// TwinCAT 3 PLC project PLC1
// Title: Sample Demo-Rack
// Company: Beckhoff Automation GmbH & Co. KG
// Author: Michael Golz
// ProjectVersion: 1.0.0
// ProgramVersion: 3.1.4026.14
// libraries:
//   Standard, * (System)
//   Tc2_Drive, * (Beckhoff Automation GmbH)
//   Tc2_EtherCAT, * (Beckhoff Automation GmbH)
//   Tc2_IoFunctions, * (Beckhoff Automation GmbH)
//   Tc2_Math, * (Beckhoff Automation GmbH)
//   Tc2_MC2, * (Beckhoff Automation GmbH)
//   Tc2_MC2_Camming, * (Beckhoff Automation GmbH)
//   Tc2_MC2_Drive, * (Beckhoff Automation GmbH)
//   Tc2_MC2_XFC, * (Beckhoff Automation GmbH)
//   Tc2_NCI, * (Beckhoff Automation GmbH)
//   Tc2_NcKinematicTransformation, * (Beckhoff Automation GmbH)
//   Tc2_PlcInterpolation, * (Beckhoff Automation GmbH)
//   Tc2_Standard, * (Beckhoff Automation GmbH)
//   Tc2_SUPS, * (Beckhoff Automation GmbH)
//   Tc2_System, * (Beckhoff Automation GmbH)
//   Tc2_Utilities, * (Beckhoff Automation GmbH)
//   Tc3_Database, * (Beckhoff Automation GmbH)
//   Tc3_EventLogger, * (Beckhoff Automation GmbH)
//   Tc3_Interfaces, * (Beckhoff Automation GmbH)
//   Tc3_IotBase, * (Beckhoff Automation GmbH)
//   Tc3_JsonXml, * (Beckhoff Automation GmbH)
//   Tc3_Module, * (Beckhoff Automation GmbH)
//   Tc3_RealtimeMonitoring, * (Beckhoff Automation GmbH)
//   TwinSafe3Diagnostics_v0.2.3, * (Beckhoff Automation LLC - Sample Code)
//   VisuDialogs, * (System)
// project tree:
//   DUTs/00_MainBlocks/ E_SystemStartupSequence.TcDUT
//   DUTs/20_Axis/ E_AxisReversingSequence.TcDUT, E_McResetStatus.TcDUT
//   DUTs/30_EtherCatDiagnostic/ E_EcDiacStatus.TcDUT, E_EcGetSlaveName.TcDUT, E_EcSystemStatus.TcDUT, ST_EcTerminalDiagInfo.TcDUT
//   DUTs/40_TwinSAFE/ ST_AdsAddr.TcDUT
//   DUTs/40_TwinSAFE/TwinSAFE_Connection/AX5805/ E_TsDiagnosisObjektsFA10AX5805.TcDUT, E_TsErrIndicesFA82AX5805.TcDUT, ST_TsControlWordAX5805.TcDUT, ST_TsDiagObjectsFA10AX5805.TcDUT, ST_TsErrIndicesFA82AX5805.TcDUT, ST_TsStatusWordAX5805.TcDUT
//   DUTs/40_TwinSAFE/TwinSAFE_Connection/EK1914/ ST_TsDiagObjectsBitsEK1914.TcDUT, ST_TsDiagObjectsEK1914.TcDUT
//   DUTs/40_TwinSAFE/TwinSAFE_Connection/EL1904/ ST_TsDiagObjectsBitsEL1904.TcDUT, ST_TsDiagObjectsEL1904.TcDUT
//   DUTs/40_TwinSAFE/TwinSAFE_Connection/EL2904/ ST_TsDiagObjectsBitsEL2904.TcDUT, ST_TsDiagObjectsEL2904.TcDUT
//   DUTs/40_TwinSAFE/TwinSAFE_Connection/ E_TsCycleDiagObj.TcDUT, ST_TsConnectionInfo1Byte.TcDUT, ST_TsConnectionInfo2Byte.TcDUT, ST_TsConnectionInfo8Byte.TcDUT, ST_TsConnectionInfoEL3214.TcDUT, ST_TsConnectionInfoEL5021.TcDUT, ST_TsSlave2Temp.TcDUT, ST_TsSlave3Temp.TcDUT
//   DUTs/40_TwinSAFE/TwinSAFE_Functionblocks/ E_TsFbType.TcDUT, ST_TsFbInfo.TcDUT
//   DUTs/40_TwinSAFE/TwinSAFE_Group/ ST_TsGroupInfo.TcDUT
//   DUTs/ E_SampleMode.TcDUT
//   / extMarkTask.TcTTO, GlobalTextList.TcGTLO, PlcTask.TcTTO, PlcTaskFast.TcTTO, Visualization Manager.TcVMO (not stored)
//   GVLs/ GVL.TcGVL, GVL00_IO_CX.TcGVL, GVL01_IO_EK1100.TcGVL, GVL02_IO_EK1101.TcGVL, GVL10_VAR_PRG.TcGVL, GVL20_Axis.TcGVL, GVL30_DiagnosticEtherCAT.TcGVL
//   POUs/Motion/ CamTable.TcPOU, Ext_SP_Gen.TcPOU, Axis1.TcPOU, AxisGeneral.TcPOU, Axis2.TcPOU, Axis3.TcPOU, Axis4.TcPOU, NCI.TcPOU
//   POUs/Database Server/ CSVSample.TcPOU, E_WriteMode.TcDUT, FB_CSV_Access.TcPOU, ST_CSVDataStruct.TcDUT
//   POUs/GeneralPlcBlocks/ FB_GenerateData.TcPOU, Blinker.TcPOU, ClockGenerator.TcPOU, GeneralPlc.TcPOU
//   POUs/IoT and JsonXml/FBs/ FB_JSONEncoding.TcPOU, FB_MqttCom_String.TcPOU, prgPopulateStructure.TcPOU
//   POUs/IoT and JsonXml/ IoTDataStruct.TcDUT, IoT_JSON_XML.TcPOU
//   POUs/MainPOUs/ MAIN.TcPOU, MAINFast.TcPOU, V_MAIN.TcVIS
//   POUs/GeneralPlcBlocks/Components/ FB_Blinker.TcPOU, F_Scaling.TcPOU
//   POUs/Motion/Components/ FB_Axis.TcPOU, FB_AxisAX5xxx.TcPOU, FB_ReversingSequence.TcPOU, MC_Reset_Ax5xxx.TcPOU
//   POUs/EtherCatDiagnostic/Components/ FB_DiagnosticEtherCAT.TcPOU
//   POUs/EtherCatDiagnostic/ DiagnosticEtherCAT.TcPOU
//   POUs/RT Monitor/ extMarksPrg.TcPOU, simpleMarksPrg.TcPOU
//   POUs/RT Monitor/logging/ ConsumeTime.TcPOU
//   POUs/Sample OOP/Cylinder/ FB_Cylinder.TcPOU, FB_CylinderDiag.TcPOU, ICylinder.TcIO
//   POUs/Sample OOP/ FB_OOPAxisTable.TcPOU, FB_OOPCylinderRegulator.TcPOU
//   POUs/Sample OOP/Regulator/ FB_BasicP.TcPOU, FB_BasicPID.TcPOU, IRegulator.TcIO, ST_RegParams.TcDUT
//   POUs/Sample OOP/Table/Axis/ FB_AX5000Axis.TcPOU, FB_NcAxis.TcPOU, IAxis.TcIO
//   POUs/Sample OOP/Table/ E_AxisState.TcDUT, E_MoveCmd.TcDUT, FB_Table.TcPOU
//   POUs/TwinSAFE/Components/ FB_EcGetSlaveName.TcPOU, FB_TwinSafeConnectionAX5805.TcPOU, FB_TwinSafeConnectionEK1914.TcPOU, FB_TwinSafeConnectionEL1904.TcPOU, FB_TwinSafeConnectionEL2904.TcPOU, FB_TwinSafeConnectionEL3214.TcPOU, FB_TwinSafeConnectionEL5021.TcPOU, FB_TwinSafeFB.TcPOU, FB_TwinSafeGroup.TcPOU, FB_TwinSafeGroupExt.TcPOU
//   POUs/TwinSAFE/ TwinSAFE.TcPOU
//   POUs/XFC/ AverageOut.TcPOU, DcTimes.TcPOU, AnalogOutputOversampling.TcPOU, PositionCamTimeStampAxis2.TcPOU, SignalLengthMeasurementCamAxis2.TcPOU, TouchProbeTimeStampCamAxis2.TcPOU
//   POUs/Sample OOP Conveyor/Axis Blocks/ FB_AX5000.TcPOU, FB_AxisNc.TcPOU, FB_Stepper.TcPOU, FB_VeryBasicMotor.TcPOU, I_Axis.TcIO
//   POUs/Sample OOP Conveyor/Device And Station Blocks/ FB_Conveyor.TcPOU, FB_Device.TcPOU, FB_Station.TcPOU, FB_TransferStation.TcPOU, GVL_Products.TcGVL, I_Mode.TcIO
//   POUs/Sample OOP Conveyor/Device And Station Blocks/Internal/ E_Modes.TcDUT, E_PartQuality.TcDUT, ST_PartData.TcDUT
//   POUs/Sample OOP Conveyor/ FB_OOPConveyor.TcPOU, V_OOP_Conveyor.TcVIS
//   POUs/Sample OOP Conveyor/Internal Visus/ Conveyor.TcVIS, ConveyorAuto.TcVIS, ConveyorData.TcVIS
//   POUs/Sample UML SC/ FB_UML_SC_Composite.TcPOU, FB_UML_SC_Lamp.TcPOU, GVL_UML.TcGVL, Visu_Composite.TcVIS, Visu_Lamp.TcVIS
//   POUs/SampleIEC Languages/Datatypes/ E_Commands.TcDUT, E_Operation.TcDUT
//   POUs/SampleIEC Languages/FunctionBlocks/ FB_CFC_SamplePOU.TcPOU, FB_CFC_SamplePouPageOriented.TcPOU, FB_FBD_IL_LD_SamplePOU.TcPOU, FB_SFC_SamplePou.TcPOU, FB_ST_SamplePOU.TcPOU
//   POUs/SampleIEC Languages/ MAIN_CFC.TcPOU, MAIN_CFC_PageOriented.TcPOU, MAIN_FBD_IL_LD.TcPOU, MAIN_SFC.TcPOU, MAIN_ST.TcPOU
//   VISUs/ MotionProfiles.TcVIS, HmiEtherCatDiagnostic.TcVIS, HmiAxisReversingSequence.TcVIS, HmiStartPage.TcVIS, HmiTwinSAFEDiagnostic.TcVIS
//   VISUs/HmiTemplatesAxis/ TplAxisControl.TcVIS, TplAxisReversingSequence.TcVIS
//   VISUs/HmiTemplatesTwinSAFE/ TplTsConnectionAX5805.TcVIS, TplTsConnectionEK1914.TcVIS, TplTsConnectionEL1904.TcVIS, TplTsConnectionEL2904.TcVIS, TplTsConnectionEL3214.TcVIS, TplTsConnectionEL5021.TcVIS, TplTsFb.TcVIS, TplTsGroup.TcVIS, TplTsGroupExt.TcVIS
// real-time tasks:
//   TASK PlcTask: cycle T#1ms, priority 8, ADS port 350
//   TASK PlcTaskFast: cycle T#100us, priority 4, ADS port 351
//   TASK VISU_TASK: cycle T#200000us, priority 30, ADS port 352
//   TASK extMarkTask: cycle T#1ms, priority 20, ADS port 353
// motion (NC):
//   TASK NC-Task 1 SAF: cycle T#1ms, priority 6, ADS port 501
//   TASK NC-Task 1 SVB: cycle T#10ms, priority 12, ADS port 511
//   AXIS Axis 1 Stepper (id 1)
//     General: UnitName=Degree
//     Dynamic: Acceleration=21600, Deceleration=21600, Jerk=259200, DelayTime=0.004
//     Velo: SlowManual=10, FastManual=150, Maximum=3600
//     OtherSettings: AllowMotionCmdToSlave=true
//     encoder EncType=4
//       EncPara: ScaleFactorNumerator=0.087890625, Inverse=true, EncMode=3, MaxCount=#xffffffff
//         Inc: RefSoftSyncMask=#x0000ffff
//     drive DrvType=24
//       DrvPara: Inverse=true
//         Analog: VeloReferenz=3600
//         TimeComp: TaskDelayCycles=1
//     controller CtrType=1
//       CtrPara: PriorControlFactor=1
//         PosDiffControl: Range=10
//         PID: PosKp=70
//         Observer: BandWidth=20
//   AXIS Axis 2 Servo EL (id 2)
//     Dynamic: Acceleration=5154.753, Deceleration=5154.753, Jerk=15464.259, DelayTime=0.004
//     Velo: RefSearch=34.36502, RefSync=34.36502, SlowManual=171.8251, FastManual=1030.9506, Fast=3436.502, Maximum=3436.502
//     OtherSettings: AllowMotionCmdToSlave=true
//     encoder EncType=19
//       EncPara: ScaleFactorNumerator=104.8576, ScaleFactorDenominator=1048576, Offset=-47.46, EncMode=3, MaxCount=#xffffffff
//     drive DrvType=16
//       DrvPara: MaxCount=#xffffffff, DriveControlDWord=#x00000100
//         Analog: VeloReferenz=3780.1522, VeloScale=32
//         TimeComp: TaskDelayCycles=1
//     controller CtrType=1
//       CtrPara: PriorControlFactor=1
//         PosDiffControl: Range=10
//         PID: PosKp=40
//         Observer: BandWidth=20
//   AXIS Axis 3 Servo A AX (id 3)
//     General: UnitName=Degree
//     Dynamic: Acceleration=108000, Deceleration=108000, Jerk=1296000
//     Velo: RefSearch=180, RefSync=180, SlowManual=10, FastManual=150, Fast=18000, Maximum=18000
//     OtherSettings: AllowMotionCmdToSlave=true
//     encoder EncType=8
//       EncPara: ScaleFactorNumerator=360, ScaleFactorDenominator=1048576, Offset=267.17, Inverse=true, MaxCount=#xffffffff
//     drive DrvType=9
//       DrvPara: Inverse=true, MaxCount=#xffffffff, DriveControlDWord=#x00030100
//         Analog: VeloReferenz=19800, VeloScale=1.02400649589962
//         TimeComp: TaskDelayCycles=1
//     controller CtrType=1
//       CtrPara: PriorControlFactor=1
//         PosDiffControl: Enable=false
//         Observer: BandWidth=20
//   AXIS Axis 4 Servo B AX (id 4)
//     General: UnitName=Degree
//     Dynamic: Acceleration=270000, Deceleration=270000, Jerk=8100000
//     Velo: RefSearch=180, RefSync=180, SlowManual=10, FastManual=150, Fast=18000, Maximum=18000
//     OtherSettings: AllowMotionCmdToSlave=true
//     encoder EncType=8
//       EncPara: ScaleFactorNumerator=360, ScaleFactorDenominator=1048576, Offset=16.16, MaxCount=#xffffffff
//     drive DrvType=9
//       DrvPara: MaxCount=#xffffffff, DriveControlDWord=#x00030100
//         Analog: VeloReferenz=19800, VeloScale=1.02400649589962
//         TimeComp: TaskDelayCycles=1
//     controller CtrType=1
//       CtrPara: PriorControlFactor=1
//         Observer: BandWidth=20
//   AXIS Axis 5 Handwheel (id 5)
//     OtherSettings: AllowMotionCmdToSlave=true
//     encoder EncType=4
//       EncPara: ScaleFactorNumerator=0.0375, Inverse=true, MaxCount=#x0000ffff
//         Inc: RefSoftSyncMask=#x0000ffff
//     drive DrvType=5
//       TimeComp: TaskDelayCycles=1
//     controller CtrType=1
//       CtrPara: PriorControlFactor=1
//         Observer: BandWidth=20
// I/O:
//   DEVICE Device 1 (EtherCAT), AmsNetId 5.77.241.156.2.1
//     Term 1 (EK1200) [EK1200-5000 EtherCAT Power supply (2A E-Bus)]
//       Term 2 (EL1008) [EL1008 8Ch. Dig. Input 24V, 3ms]
//       Term 3 (EL2008) [EL2008 8Ch. Dig. Output 24V, 0.5A]
//       Term 4 (EL5151) [EL5151 1Ch. Inc. Encoder]
//       Term 5 (EL9110) [EL9110 Power Supplier with LED (24V, Diagnostics)]
//       Term 6 (EL9576) [EL9576 Brake chopper terminal]
//       Term 7 (EL7037) [EL7037 1Ch. Stepper motor output stage (24V, 1.5A)]
//       Term 8 (EL9512) [EL9512 Power supply terminal 12V]
//       Term 9 (EL3162) [EL3162 2Ch. Ana. Input 0-10V]
//       Term 10 (EL4102) [EL4102 2Ch. Ana. Output  0-10V, 16bit]
//       Term 11 (EL6900) [EL6900, TwinSAFE PLC] (disabled)
//       Term 43 (EL6910) [EL6910, TwinSAFE PLC]
//       Term 12 (EK1122) [EK1122 2 port EtherCAT junction]
//         Drive 29 (AX5203-0000-0215)_1 [AX5203-0000-0215 EtherCAT Drive (SoE, 2 Ch.)]
//           Term 34 (AX5805) [AX5805 (Safety Drive Option)]
//             modules: Module 1 (Safety Process Data, 2 axis), Module 2 (Standard Process Data, 2 axis)
//         Term 13 (EK1100) [EK1100 EtherCAT Coupler (2A E-Bus)]
//           Term 14 (EL1859) [EL1859 8Ch. Dig. Input 24V, 3ms, 8Ch. Dig. Output 24V, 0.5A]
//           Term 15 (EL1904) [EL1904, 4 Ch. Safety Input 24V, TwinSAFE]
//             modules: Module 1 (FSOES)
//           Term 16 (EL2904) [EL2904, 4 Ch. Safety Output 24V, 0.5A, TwinSAFE]
//             modules: Module 1 (FSOES), Module 2 (DO)
//           Term 17 (EL9110) [EL9110 Power Supplier with LED (24V, Diagnostics)]
//           Term 18 (EL2004) [EL2004 4Ch. Dig. Output 24V, 0.5A]
//           Term 19 (EL9410) [EL9410 E-Bus Power Supplier  (Diagnostics)]
//           Term 20 (EL7201-0010) [EL7201-0010 1Ch. MDP742 Servo motor output stage with OCT (50V, 4A)]
//             startup 32784:18 := 0500
//             startup 32784:19 := B200
//             startup 32784:20 := 96000000 // Velocity loop integral time
//             startup 32784:21 := 2B000000 // Velocity loop proportional gain
//             startup 32785:17 := 98210000
//             startup 32785:18 := 960A0000
//             startup 32785:19 := 03
//             startup 32785:21 := 0E01
//             startup 32785:22 := 46000000
//             startup 32785:24 := 21000000
//             startup 32785:25 := 0F00
//             startup 32785:27 := 4F060000
//             startup 32785:45 := 5501
//           Term 30 (EL9011) [EL9011 End Terminal]
//     Term 21 (EK1101) [EK1101 EtherCAT Coupler (2A E-Bus, ID switch)]
//       Term 22 (EL1904) [EL1904, 4 Ch. Safety Input 24V, TwinSAFE]
//         modules: Module 1 (FSOES)
//       Term 23 (EL1252) [EL1252 2Ch. Fast Dig. Input 24V, 1µs, DC Latch]
//       Term 24 (EL1262) [EL1262 2Ch. Dig. Input 24V, 1µs, DC Oversample]
//       Term 25 (EL2252) [EL2252 2Ch. Dig. Output 24V, 0.5A, DC Time Stamp]
//       Term 26 (EL3702) [EL3702 2Ch. Ana. Input +/-10V, DIFF, Oversample]
//       Term 27 (EL4732) [EL4732 2Ch. Ana. Output +/-10V, Oversample]
//       Term 28 (EL2004) [EL2004 4Ch. Dig. Output 24V, 0.5A]
//       Term 31 (EL9011) [EL9011 End Terminal]
// variable links:
//   Device 1 (EtherCAT) <-> Device 1 (EtherCAT)/Term 1 (EK1200)/Term 43 (EL6910)
//     Term 1 (EK1200)/Term 12 (EK1122)/Drive 29 (AX5203-0000-0215)_1/Term 34 (AX5805)/Module 1 (Safety Process Data, 2 axis)/Inputs (Statusword)/FSOE <-> ConnectionOutputs/Message_5 RxPDO
//     Term 1 (EK1200)/Term 12 (EK1122)/Drive 29 (AX5203-0000-0215)_1/Term 34 (AX5805)/Module 1 (Safety Process Data, 2 axis)/Outputs (Controlword)/FSOE <-> ConnectionInputs/Message_5 TxPDO
//     Term 1 (EK1200)/Term 12 (EK1122)/Term 13 (EK1100)/Term 15 (EL1904)/Module 1 (FSOES)/RxPDO/FSOE <-> ConnectionInputs/Message_2 TxPDO
//     Term 1 (EK1200)/Term 12 (EK1122)/Term 13 (EK1100)/Term 16 (EL2904)/Module 1 (FSOES)/RxPDO/FSOE <-> ConnectionInputs/Message_3 TxPDO
//     Term 1 (EK1200)/Term 12 (EK1122)/Term 13 (EK1100)/Term 15 (EL1904)/Module 1 (FSOES)/TxPDO/FSOE <-> ConnectionOutputs/Message_2 RxPDO
//     Term 1 (EK1200)/Term 12 (EK1122)/Term 13 (EK1100)/Term 16 (EL2904)/Module 1 (FSOES)/TxPDO/FSOE <-> ConnectionOutputs/Message_3 RxPDO
//     Term 21 (EK1101)/Term 22 (EL1904)/Module 1 (FSOES)/RxPDO/FSOE <-> ConnectionInputs/Message_4 TxPDO
//     Term 21 (EK1101)/Term 22 (EL1904)/Module 1 (FSOES)/TxPDO/FSOE <-> ConnectionOutputs/Message_4 RxPDO
//   NC-Task 1 SAF/Axes/Axis 1 Stepper <-> Device 1 (EtherCAT)/Term 1 (EK1200)/Term 7 (EL7037)
//     Drive/Inputs/In/nState1 @bit 3 <-> STM Status/Status/Error
//     Drive/Inputs/In/nState1 @bit 7 <-> STM Status/Status/Motor stall
//     Drive/Inputs/In/nState1 @bit 5 <-> STM Status/Status/Moving negative
//     Drive/Inputs/In/nState1 @bit 4 <-> STM Status/Status/Moving positive
//     Drive/Inputs/In/nState1 @bit 1 <-> STM Status/Status/Ready
//     Drive/Inputs/In/nState1 <-> STM Status/Status/Ready to enable
//     Drive/Inputs/In/nState1 @bit 6 <-> STM Status/Status/Torque reduced
//     Drive/Inputs/In/nState1 @bit 2 <-> STM Status/Status/Warning
//     Drive/Inputs/In/nState2 @bit 3 <-> STM Status/Status/Digital input 1
//     Drive/Inputs/In/nState2 @bit 4 <-> STM Status/Status/Digital input 2
//     Drive/Inputs/In/nState2 @bit 5 <-> STM Status/Status/Sync error
//     Drive/Inputs/In/nState2 @bit 7 <-> STM Status/Status/TxPDO Toggle
//     Drive/Inputs/In/nState4 @bit 1 <-> WcState/InputToggle
//     Drive/Inputs/In/nState4 <-> WcState/WcState
//     Drive/Outputs/Out/nCtrl1 <-> STM Control/Control/Enable
//     Drive/Outputs/Out/nCtrl1 @bit 2 <-> STM Control/Control/Reduce torque
//     Drive/Outputs/Out/nCtrl1 @bit 1 <-> STM Control/Control/Reset
//     Drive/Outputs/Out/nCtrl2 @bit 3 <-> STM Control/Control/Digital output 1
//     Drive/Outputs/Out/nDataOut2[0] <-> STM Velocity/Velocity
//     Enc/Inputs/In/nDataIn1 <-> ENC Status/Counter value
//     Enc/Inputs/In/nDataIn2 <-> ENC Status/Latch value
//     Enc/Inputs/In/nState1 @bit 4 <-> ENC Status/Status/Counter overflow
//     Enc/Inputs/In/nState1 @bit 3 <-> ENC Status/Status/Counter underflow
//     Enc/Inputs/In/nState1 @bit 7 <-> ENC Status/Status/Extrapolation stall
//     Enc/Inputs/In/nState1 <-> ENC Status/Status/Latch C valid
//     Enc/Inputs/In/nState1 @bit 1 <-> ENC Status/Status/Latch extern valid
//     Enc/Inputs/In/nState1 @bit 2 <-> ENC Status/Status/Set counter done
//     Enc/Inputs/In/nState2 @bit 4 <-> ENC Status/Status/Status of extern latch
//     Enc/Inputs/In/nState2 <-> ENC Status/Status/Status of input A
//     Enc/Inputs/In/nState2 @bit 1 <-> ENC Status/Status/Status of input B
//     Enc/Inputs/In/nState2 @bit 2 <-> ENC Status/Status/Status of input C
//     Enc/Inputs/In/nState2 @bit 5 <-> ENC Status/Status/Sync error
//     Enc/Inputs/In/nState2 @bit 7 <-> ENC Status/Status/TxPDO Toggle
//     Enc/Inputs/In/nState4 @bit 1 <-> WcState/InputToggle
//     Enc/Inputs/In/nState4 <-> WcState/WcState
//     Enc/Outputs/Out/nCtrl1 <-> ENC Control/Control/Enable latch C
//     Enc/Outputs/Out/nCtrl1 @bit 3 <-> ENC Control/Control/Enable latch extern on negative edge
//     Enc/Outputs/Out/nCtrl1 @bit 1 <-> ENC Control/Control/Enable latch extern on positive edge
//     Enc/Outputs/Out/nCtrl1 @bit 2 <-> ENC Control/Control/Set counter
//     Enc/Outputs/Out/nDataOut1 <-> ENC Control/Set counter value
//   NC-Task 1 SAF/Axes/Axis 2 Servo EL <-> Device 1 (EtherCAT)/Term 1 (EK1200)/Term 12 (EK1122)/Term 13 (EK1100)/Term 20 (EL7201-0010)
//     Drive/Inputs/In/nDataIn1 <-> DRV Following error actual value/Following error actual value
//     Drive/Inputs/In/nDataIn3[0] <-> DRV Torque actual value/Torque actual value
//     Drive/Inputs/In/nDcOutputTime <-> InfoData/DcOutputShift
//     Drive/Inputs/In/nState1 <-> DRV Statusword/Statusword
//     Drive/Inputs/In/nState2 <-> DRV Statusword/Statusword @bit 8
//     Drive/Inputs/In/nState4 @bit 1 <-> WcState/InputToggle
//     Drive/Inputs/In/nState4 <-> WcState/WcState
//     Drive/Outputs/Out/nCtrl1 <-> DRV Controlword/Controlword
//     Drive/Outputs/Out/nCtrl2 <-> DRV Controlword/Controlword @bit 8
//     Drive/Outputs/Out/nDataOut1 <-> DRV Target position/Target position
//     Drive/Outputs/Out/nDataOut2 <-> DRV Target velocity/Target velocity
//     Enc/Inputs/In/nDataIn1 <-> FB Position/Position
//     Enc/Inputs/In/nDcInputTime <-> InfoData/DcInputShift
//     Enc/Inputs/In/nState4 @bit 1 <-> WcState/InputToggle
//     Enc/Inputs/In/nState4 <-> WcState/WcState
//     Enc/Inputs/In/nState5 <-> FB Touch probe status/Touch probe status/TP1 Enable
//     Enc/Inputs/In/nState6 <-> FB Touch probe status/Touch probe status/TP2 Enable
//     Enc/Inputs/In/nState5 @bit 7 <-> FB Touch probe status/Touch probe status/TP1 Input
//     Enc/Inputs/In/nState6 @bit 7 <-> FB Touch probe status/Touch probe status/TP2 Input
//     Enc/Inputs/In/nState5 @bit 2 <-> FB Touch probe status/Touch probe status/TP1 Neg value stored
//     Enc/Inputs/In/nState6 @bit 2 <-> FB Touch probe status/Touch probe status/TP2 Neg value stored
//     Enc/Inputs/In/nState5 @bit 1 <-> FB Touch probe status/Touch probe status/TP1 Pos value stored
//     Enc/Inputs/In/nState6 @bit 1 <-> FB Touch probe status/Touch probe status/TP2 Pos value stored
//   NC-Task 1 SAF/Axes/Axis 3 Servo A AX <-> Device 1 (EtherCAT)/Term 1 (EK1200)/Term 12 (EK1122)/Drive 29 (AX5203-0000-0215)_1
//     Drive/Inputs/In/nDataIn1 <-> AT 1/Following distance
//     Drive/Inputs/In/nDcOutputTime <-> InfoData/DcOutputShift
//     Drive/Inputs/In/nState1 <-> AT 1/Drive status word @bit 8
//     Drive/Inputs/In/nState2 <-> AT 1/Drive status word
//     Drive/Inputs/In/nState4 @bit 1 <-> WcState/InputToggle
//     Drive/Outputs/Out/nCtrl1 <-> MDT 1/Master control word @bit 8
//     Drive/Outputs/Out/nDataOut1 <-> MDT 1/Position command value
//     Enc/Inputs/In/nDataIn1 <-> AT 1/Position feedback 1 value
//     Enc/Inputs/In/nDcInputTime <-> InfoData/DcInputShift
//     Enc/Inputs/In/nState4 @bit 1 <-> WcState/InputToggle
//   NC-Task 1 SAF/Axes/Axis 4 Servo B AX <-> Device 1 (EtherCAT)/Term 1 (EK1200)/Term 12 (EK1122)/Drive 29 (AX5203-0000-0215)_1
//     Drive/Inputs/In/nDataIn1 <-> AT 2/Following distance
//     Drive/Inputs/In/nDcOutputTime <-> InfoData/DcOutputShift
//     Drive/Inputs/In/nState1 <-> AT 2/Drive status word @bit 8
//     Drive/Inputs/In/nState2 <-> AT 2/Drive status word
//     Drive/Inputs/In/nState4 @bit 1 <-> WcState/InputToggle
//     Drive/Outputs/Out/nCtrl1 <-> MDT 2/Master control word @bit 8
//     Drive/Outputs/Out/nDataOut1 <-> MDT 2/Position command value
//     Enc/Inputs/In/nDataIn1 <-> AT 2/Position feedback 1 value
//     Enc/Inputs/In/nDcInputTime <-> InfoData/DcInputShift
//     Enc/Inputs/In/nState4 @bit 1 <-> WcState/InputToggle
//   NC-Task 1 SAF/Axes/Axis 5 Handwheel <-> Device 1 (EtherCAT)/Term 1 (EK1200)/Term 4 (EL5151)
//     Enc/Inputs/In/nDataIn1[0] <-> ENC Inputs/Counter value
//     Enc/Inputs/In/nDataIn2[0] <-> ENC Inputs/Latch value
//     Enc/Inputs/In/nState1 @bit 7 <-> ENC Inputs/Status/Extrapolation stall
//     Enc/Inputs/In/nState1 <-> ENC Inputs/Status/Latch C valid
//     Enc/Inputs/In/nState1 @bit 1 <-> ENC Inputs/Status/Latch extern valid
//     Enc/Inputs/In/nState1 @bit 2 <-> ENC Inputs/Status/Set counter done
//     Enc/Inputs/In/nState2 @bit 4 <-> ENC Inputs/Status/Status of extern latch
//     Enc/Inputs/In/nState2 <-> ENC Inputs/Status/Status of input A
//     Enc/Inputs/In/nState2 @bit 1 <-> ENC Inputs/Status/Status of input B
//     Enc/Inputs/In/nState2 @bit 2 <-> ENC Inputs/Status/Status of input C
//     Enc/Inputs/In/nState2 @bit 5 <-> ENC Inputs/Status/Sync error
//     Enc/Inputs/In/nState2 @bit 7 <-> ENC Inputs/Status/TxPDO Toggle
//     Enc/Inputs/In/nState4 @bit 1 <-> WcState/InputToggle
//     Enc/Inputs/In/nState4 <-> WcState/WcState
//     Enc/Outputs/Out/nCtrl1 <-> ENC Outputs/Control/Enable latch C
//     Enc/Outputs/Out/nCtrl1 @bit 3 <-> ENC Outputs/Control/Enable latch extern on negative edge
//     Enc/Outputs/Out/nCtrl1 @bit 1 <-> ENC Outputs/Control/Enable latch extern on positive edge
//     Enc/Outputs/Out/nCtrl1 @bit 2 <-> ENC Outputs/Control/Set counter
//     Enc/Outputs/Out/nDataOut1[0] <-> ENC Outputs/Set counter value
//   PLC1/PLC1 Instance <-> Device 1 (EtherCAT)
//     PlcTask Inputs/GVL30_DiagnosticEtherCAT.fbDiagnosticEtherCAT.cbAmsNetId <-> InfoData/AmsNetId
//     PlcTask Inputs/GVL30_DiagnosticEtherCAT.fbDiagnosticEtherCAT.nCfgSlaveCount <-> InfoData/CfgSlaveCount
//     PlcTask Inputs/GVL30_DiagnosticEtherCAT.fbDiagnosticEtherCAT.nDevId <-> InfoData/DevId
//     PlcTask Inputs/GVL30_DiagnosticEtherCAT.fbDiagnosticEtherCAT.nDevState <-> Inputs/DevState
//     PlcTask Inputs/GVL30_DiagnosticEtherCAT.fbDiagnosticEtherCAT.nFrmXWcState[0] <-> Inputs/Frm0WcState
//   PLC1/PLC1 Instance <-> Device 1 (EtherCAT)/Term 1 (EK1200)/Term 10 (EL4102)
//     PlcTask Outputs/GVL00_IO_CX.nAnalogOutP10 <-> Channel 1/Output
//     PlcTaskFast Outputs/GVL00_IO_CX.nAnalogOutP11 <-> Channel 2/Output
//   PLC1/PLC1 Instance <-> Device 1 (EtherCAT)/Term 1 (EK1200)/Term 12 (EK1122)/Drive 29 (AX5203-0000-0215)_1
//     PlcTask Inputs/GVL20_Axis.nAX5203DigitalInputs <-> AT 1/Digital inputs, state
//     PlcTask Inputs/GVL20_Axis.nAxis3TorqueFeedback <-> AT 1/Torque/force feedback value
//     PlcTask Inputs/GVL20_Axis.nAxis4TorqueFeedback <-> AT 2/Torque/force feedback value
//     PlcTask Outputs/GVL20_Axis.nAX5203DigitalOutputs <-> MDT 1/Digital outputs
//   PLC1/PLC1 Instance <-> Device 1 (EtherCAT)/Term 1 (EK1200)/Term 12 (EK1122)/Term 13 (EK1100)/Term 14 (EL1859)
//     PlcTask Inputs/GVL01_IO_EK1100.bAxis2ReferenceCamEL1 <-> Channel 5/Input
//     PlcTask Inputs/GVL01_IO_EK1100.bSwitchS20 <-> Channel 1/Input
//     PlcTask Inputs/GVL01_IO_EK1100.bSwitchS21 <-> Channel 2/Input
//     PlcTask Inputs/GVL01_IO_EK1100.bSwitchS22 <-> Channel 3/Input
//     PlcTask Inputs/GVL01_IO_EK1100.bSwitchS31 <-> Channel 4/Input
//     PlcTask Outputs/GVL01_IO_EK1100.bLedH23 <-> Channel 13/Output
//     PlcTask Outputs/GVL01_IO_EK1100.bLedH24 <-> Channel 14/Output
//     PlcTask Outputs/GVL01_IO_EK1100.bLedH25 <-> Channel 15/Output
//     PlcTask Outputs/GVL01_IO_EK1100.bLedH26 <-> Channel 16/Output
//     PlcTask Outputs/GVL01_IO_EK1100.bLedH31 <-> Channel 9/Output
//     PlcTask Outputs/GVL01_IO_EK1100.bLedH32 <-> Channel 10/Output
//     PlcTask Outputs/GVL01_IO_EK1100.bLedH33 <-> Channel 11/Output
//   PLC1/PLC1 Instance <-> Device 1 (EtherCAT)/Term 1 (EK1200)/Term 12 (EK1122)/Term 13 (EK1100)/Term 15 (EL1904)
//     PlcTask Inputs/TwinSAFE.fbSafeConnectionEL1904_1_Group1.nEcSlaveState <-> InfoData/State
//     PlcTask Inputs/TwinSAFE.fbSafeConnectionEL1904_1_Group1.stEcAdsAddr <-> InfoData/AdsAddr
//   PLC1/PLC1 Instance <-> Device 1 (EtherCAT)/Term 1 (EK1200)/Term 12 (EK1122)/Term 13 (EK1100)/Term 16 (EL2904)
//     PlcTask Inputs/TwinSAFE.fbSafeConnectionEL2904_1_Group1.nEcSlaveState <-> InfoData/State
//     PlcTask Inputs/TwinSAFE.fbSafeConnectionEL2904_1_Group1.stEcAdsAddr <-> InfoData/AdsAddr
//   PLC1/PLC1 Instance <-> Device 1 (EtherCAT)/Term 1 (EK1200)/Term 12 (EK1122)/Term 13 (EK1100)/Term 17 (EL9110)
//     PlcTask Inputs/GVL01_IO_EK1100.bPotentialConduktorK124VOk <-> PowerOK/Input
//   PLC1/PLC1 Instance <-> Device 1 (EtherCAT)/Term 1 (EK1200)/Term 12 (EK1122)/Term 13 (EK1100)/Term 18 (EL2004)
//     PlcTask Outputs/GVL01_IO_EK1100.bLedH20 <-> Channel 1/Output
//     PlcTask Outputs/GVL01_IO_EK1100.bLedH21 <-> Channel 2/Output
//     PlcTask Outputs/GVL01_IO_EK1100.bLedH22 <-> Channel 3/Output
//   PLC1/PLC1 Instance <-> Device 1 (EtherCAT)/Term 1 (EK1200)/Term 12 (EK1122)/Term 13 (EK1100)/Term 19 (EL9410)
//     PlcTask Inputs/GVL01_IO_EK1100.bPotentialEBusUs24VNotOk <-> Status Us/Undervoltage
//     PlcTask Inputs/GVL01_IO_EK1100.bPotentialServoUp24VNotOk <-> Status Up/Undervoltage
//   PLC1/PLC1 Instance <-> Device 1 (EtherCAT)/Term 1 (EK1200)/Term 2 (EL1008)
//     PlcTask Inputs/GVL00_IO_CX.bSwitchS10 <-> Channel 1/Input
//     PlcTask Inputs/GVL00_IO_CX.bSwitchS11 <-> Channel 2/Input
//     PlcTask Inputs/GVL00_IO_CX.bSwitchS12 <-> Channel 3/Input
//     PlcTask Inputs/GVL00_IO_CX.bSwitchS13 <-> Channel 4/Input
//     PlcTask Inputs/GVL00_IO_CX.bSwitchS14 <-> Channel 5/Input
//     PlcTask Inputs/GVL00_IO_CX.bSwitchS15 <-> Channel 6/Input
//     PlcTask Inputs/GVL00_IO_CX.bSwitchS16 <-> Channel 7/Input
//     PlcTask Inputs/GVL00_IO_CX.bSwitchS17 <-> Channel 8/Input
//   PLC1/PLC1 Instance <-> Device 1 (EtherCAT)/Term 1 (EK1200)/Term 3 (EL2008)
//     PlcTask Outputs/GVL00_IO_CX.bLedH10 <-> Channel 1/Output
//     PlcTask Outputs/GVL00_IO_CX.bLedH11 <-> Channel 2/Output
//     PlcTask Outputs/GVL00_IO_CX.bLedH12 <-> Channel 3/Output
//     PlcTask Outputs/GVL00_IO_CX.bLedH13 <-> Channel 4/Output
//     PlcTask Outputs/GVL00_IO_CX.bLedH14 <-> Channel 5/Output
//     PlcTask Outputs/GVL00_IO_CX.bLedH15 <-> Channel 6/Output
//     PlcTask Outputs/GVL00_IO_CX.bLedH16 <-> Channel 7/Output
//     PlcTask Outputs/GVL00_IO_CX.bLedH17 <-> Channel 8/Output
//   PLC1/PLC1 Instance <-> Device 1 (EtherCAT)/Term 1 (EK1200)/Term 4 (EL5151)
//     PlcTask Inputs/GVL00_IO_CX.bHandwheelSwitchS28 <-> ENC Inputs/Status/Status of extern latch
//     PlcTask Inputs/GVL00_IO_CX.nHandwheelCounter <-> ENC Inputs/Counter value
//   PLC1/PLC1 Instance <-> Device 1 (EtherCAT)/Term 1 (EK1200)/Term 5 (EL9110)
//     PlcTask Inputs/GVL00_IO_CX.bPotentialStepper24VOk <-> PowerOK/Input
//   PLC1/PLC1 Instance <-> Device 1 (EtherCAT)/Term 1 (EK1200)/Term 7 (EL7037)
//     PlcTask Inputs/GVL00_IO_CX.bStepperReferenceCam <-> ENC Status/Status/Status of extern latch
//     PlcTask Inputs/GVL00_IO_CX.bSwitchS23 <-> STM Status/Status/Digital input 1
//     PlcTask Inputs/GVL00_IO_CX.bSwitchS24 <-> STM Status/Status/Digital input 2
//   PLC1/PLC1 Instance <-> Device 1 (EtherCAT)/Term 1 (EK1200)/Term 8 (EL9512)
//     PlcTask Inputs/GVL00_IO_CX.bPotentialAnalog12VOk <-> Status Uo/Power OK
//   PLC1/PLC1 Instance <-> Device 1 (EtherCAT)/Term 1 (EK1200)/Term 9 (EL3162)
//     PlcTask Inputs/GVL00_IO_CX.nAnalogInFromEL4102Out1 <-> AI Standard Channel 2/Value
//     PlcTask Inputs/GVL00_IO_CX.nAnalogInR10 <-> AI Standard Channel 1/Value
//   PLC1/PLC1 Instance <-> Device 1 (EtherCAT)/Term 21 (EK1101)/Term 22 (EL1904)
//     PlcTask Inputs/TwinSAFE.fbSafeConnectionEL1904_2_Group1.nEcSlaveState <-> InfoData/State
//     PlcTask Inputs/TwinSAFE.fbSafeConnectionEL1904_2_Group1.stEcAdsAddr <-> InfoData/AdsAddr
//   PLC1/PLC1 Instance <-> Device 1 (EtherCAT)/Term 21 (EK1101)/Term 23 (EL1252)
//     PlcTask Inputs/GVL02_IO_EK1101.stEL1252Ch1.Input <-> Channel 1/Input
//     PlcTask Inputs/GVL02_IO_EK1101.stEL1252Ch2.Input <-> Channel 2/Input
//     PlcTask Inputs/GVL02_IO_EK1101.stEL1252Ch1.Status <-> Latch/Status1
//     PlcTask Inputs/GVL02_IO_EK1101.stEL1252Ch2.Status <-> Latch/Status2
//     PlcTask Inputs/GVL02_IO_EK1101.stEL1252Ch1.TimeStampNeg <-> Latch/LatchNeg1
//     PlcTask Inputs/GVL02_IO_EK1101.stEL1252Ch2.TimeStampNeg <-> Latch/LatchNeg2
//     PlcTask Inputs/GVL02_IO_EK1101.stEL1252Ch1.TimeStampPos <-> Latch/LatchPos1
//     PlcTask Inputs/GVL02_IO_EK1101.stEL1252Ch2.TimeStampPos <-> Latch/LatchPos2
//   PLC1/PLC1 Instance <-> Device 1 (EtherCAT)/Term 21 (EK1101)/Term 24 (EL1262)
//     PlcTask Inputs/GVL02_IO_EK1101.aAxis2RefCamOs[0] <-> Ch1 Input 0/Ch1 Input
//     PlcTask Inputs/GVL02_IO_EK1101.aAxis2RefCamOs[1] <-> Ch1 Input 1/Ch1 Input
//     PlcTask Inputs/GVL02_IO_EK1101.aAxis2RefCamOs[2] <-> Ch1 Input 2/Ch1 Input
//     PlcTask Inputs/GVL02_IO_EK1101.aAxis2RefCamOs[3] <-> Ch1 Input 3/Ch1 Input
//     PlcTask Inputs/GVL02_IO_EK1101.aAxis2RefCamOs[4] <-> Ch1 Input 4/Ch1 Input
//     PlcTask Inputs/GVL02_IO_EK1101.aAxis2RefCamOs[5] <-> Ch1 Input 5/Ch1 Input
//     PlcTask Inputs/GVL02_IO_EK1101.aAxis2RefCamOs[6] <-> Ch1 Input 6/Ch1 Input
//     PlcTask Inputs/GVL02_IO_EK1101.aAxis2RefCamOs[7] <-> Ch1 Input 7/Ch1 Input
//     PlcTask Inputs/GVL02_IO_EK1101.aAxis2RefCamOs[8] <-> Ch1 Input 8/Ch1 Input
//     PlcTask Inputs/GVL02_IO_EK1101.aAxis2RefCamOs[9] <-> Ch1 Input 9/Ch1 Input
//     PlcTask Inputs/GVL02_IO_EK1101.aOsInputFromEL2252Out2[0] <-> Ch2 Input 0/Ch2 Input
//     PlcTask Inputs/GVL02_IO_EK1101.aOsInputFromEL2252Out2[1] <-> Ch2 Input 1/Ch2 Input
//     PlcTask Inputs/GVL02_IO_EK1101.aOsInputFromEL2252Out2[2] <-> Ch2 Input 2/Ch2 Input
//     PlcTask Inputs/GVL02_IO_EK1101.aOsInputFromEL2252Out2[3] <-> Ch2 Input 3/Ch2 Input
//     PlcTask Inputs/GVL02_IO_EK1101.aOsInputFromEL2252Out2[4] <-> Ch2 Input 4/Ch2 Input
//     PlcTask Inputs/GVL02_IO_EK1101.aOsInputFromEL2252Out2[5] <-> Ch2 Input 5/Ch2 Input
//     PlcTask Inputs/GVL02_IO_EK1101.aOsInputFromEL2252Out2[6] <-> Ch2 Input 6/Ch2 Input
//     PlcTask Inputs/GVL02_IO_EK1101.aOsInputFromEL2252Out2[7] <-> Ch2 Input 7/Ch2 Input
//     PlcTask Inputs/GVL02_IO_EK1101.aOsInputFromEL2252Out2[8] <-> Ch2 Input 8/Ch2 Input
//     PlcTask Inputs/GVL02_IO_EK1101.aOsInputFromEL2252Out2[9] <-> Ch2 Input 9/Ch2 Input
//     PlcTask Inputs/GVL02_IO_EK1101.nEL1262Ch1CycleCount <-> Ch1 CycleCount/Ch1 CycleCount
//     PlcTask Inputs/GVL02_IO_EK1101.nEL1262Ch2CycleCount <-> Ch2 CycleCount/Ch2 CycleCount
//   PLC1/PLC1 Instance <-> Device 1 (EtherCAT)/Term 21 (EK1101)/Term 25 (EL2252)
//     PlcTask Outputs/GVL02_IO_EK1101.stEL2252.Activate <-> DC Sync Activate/Activate
//     PlcTask Outputs/GVL02_IO_EK1101.stEL2252.Output1 <-> Channel 1/Output
//     PlcTask Outputs/GVL02_IO_EK1101.stEL2252.Output2 <-> Channel 2/Output
//     PlcTask Outputs/GVL02_IO_EK1101.stEL2252.StartTime <-> DC Sync Start/StartTime
//     PlcTask Outputs/GVL02_IO_EK1101.stEL2252.TriState1 <-> Channel 1/TriState
//     PlcTask Outputs/GVL02_IO_EK1101.stEL2252.TriState2 <-> Channel 2/TriState
//   PLC1/PLC1 Instance <-> Device 1 (EtherCAT)/Term 21 (EK1101)/Term 26 (EL3702)
//     PlcTask Inputs/GVL02_IO_EK1101.nEL3702Ch1CycleCount <-> Ch1 CycleCount/Ch1 CycleCount
//     PlcTask Inputs/GVL02_IO_EK1101.nEL3702Ch2CycleCount <-> Ch2 CycleCount/Ch2 CycleCount
//     PlcTaskFast Inputs/GVL02_IO_EK1101.aOsAnalogInR11[0] <-> Ch1 Sample 0/Ch1 Value
//     PlcTaskFast Inputs/GVL02_IO_EK1101.aOsAnalogInR11[1] <-> Ch1 Sample 1/Ch1 Value
//     PlcTaskFast Inputs/GVL02_IO_EK1101.aOsAnalogInR11[2] <-> Ch1 Sample 2/Ch1 Value
//     PlcTaskFast Inputs/GVL02_IO_EK1101.aOsAnalogInR11[3] <-> Ch1 Sample 3/Ch1 Value
//     PlcTaskFast Inputs/GVL02_IO_EK1101.aOsAnalogInR11[4] <-> Ch1 Sample 4/Ch1 Value
//     PlcTaskFast Inputs/GVL02_IO_EK1101.aOsAnalogInR11[5] <-> Ch1 Sample 5/Ch1 Value
//     PlcTaskFast Inputs/GVL02_IO_EK1101.aOsAnalogInR11[6] <-> Ch1 Sample 6/Ch1 Value
//     PlcTaskFast Inputs/GVL02_IO_EK1101.aOsAnalogInR11[7] <-> Ch1 Sample 7/Ch1 Value
//     PlcTaskFast Inputs/GVL02_IO_EK1101.aOsAnalogInR11[8] <-> Ch1 Sample 8/Ch1 Value
//     PlcTaskFast Inputs/GVL02_IO_EK1101.aOsAnalogInR11[9] <-> Ch1 Sample 9/Ch1 Value
//     PlcTaskFast Inputs/GVL02_IO_EK1101.aOsInputFromEL4732Out1[0] <-> Ch2 Sample 0/Ch2 Value
//     PlcTaskFast Inputs/GVL02_IO_EK1101.aOsInputFromEL4732Out1[1] <-> Ch2 Sample 1/Ch2 Value
//     PlcTaskFast Inputs/GVL02_IO_EK1101.aOsInputFromEL4732Out1[2] <-> Ch2 Sample 2/Ch2 Value
//     PlcTaskFast Inputs/GVL02_IO_EK1101.aOsInputFromEL4732Out1[3] <-> Ch2 Sample 3/Ch2 Value
//     PlcTaskFast Inputs/GVL02_IO_EK1101.aOsInputFromEL4732Out1[4] <-> Ch2 Sample 4/Ch2 Value
//     PlcTaskFast Inputs/GVL02_IO_EK1101.aOsInputFromEL4732Out1[5] <-> Ch2 Sample 5/Ch2 Value
//     PlcTaskFast Inputs/GVL02_IO_EK1101.aOsInputFromEL4732Out1[6] <-> Ch2 Sample 6/Ch2 Value
//     PlcTaskFast Inputs/GVL02_IO_EK1101.aOsInputFromEL4732Out1[7] <-> Ch2 Sample 7/Ch2 Value
//     PlcTaskFast Inputs/GVL02_IO_EK1101.aOsInputFromEL4732Out1[8] <-> Ch2 Sample 8/Ch2 Value
//     PlcTaskFast Inputs/GVL02_IO_EK1101.aOsInputFromEL4732Out1[9] <-> Ch2 Sample 9/Ch2 Value
//   PLC1/PLC1 Instance <-> Device 1 (EtherCAT)/Term 21 (EK1101)/Term 27 (EL4732)
//     PlcTask Outputs/GVL02_IO_EK1101.aOsOutputToEL3702In2[0] <-> Ch1 Sample 0/Ch1 Value
//     PlcTask Outputs/GVL02_IO_EK1101.aOsOutputToEL3702In2[10] <-> Ch1 Sample 10/Ch1 Value
//     PlcTask Outputs/GVL02_IO_EK1101.aOsOutputToEL3702In2[11] <-> Ch1 Sample 11/Ch1 Value
//     PlcTask Outputs/GVL02_IO_EK1101.aOsOutputToEL3702In2[12] <-> Ch1 Sample 12/Ch1 Value
//     PlcTask Outputs/GVL02_IO_EK1101.aOsOutputToEL3702In2[13] <-> Ch1 Sample 13/Ch1 Value
//     PlcTask Outputs/GVL02_IO_EK1101.aOsOutputToEL3702In2[14] <-> Ch1 Sample 14/Ch1 Value
//     PlcTask Outputs/GVL02_IO_EK1101.aOsOutputToEL3702In2[15] <-> Ch1 Sample 15/Ch1 Value
//     PlcTask Outputs/GVL02_IO_EK1101.aOsOutputToEL3702In2[16] <-> Ch1 Sample 16/Ch1 Value
//     PlcTask Outputs/GVL02_IO_EK1101.aOsOutputToEL3702In2[17] <-> Ch1 Sample 17/Ch1 Value
//     PlcTask Outputs/GVL02_IO_EK1101.aOsOutputToEL3702In2[18] <-> Ch1 Sample 18/Ch1 Value
//     PlcTask Outputs/GVL02_IO_EK1101.aOsOutputToEL3702In2[19] <-> Ch1 Sample 19/Ch1 Value
//     PlcTask Outputs/GVL02_IO_EK1101.aOsOutputToEL3702In2[1] <-> Ch1 Sample 1/Ch1 Value
//     PlcTask Outputs/GVL02_IO_EK1101.aOsOutputToEL3702In2[20] <-> Ch1 Sample 20/Ch1 Value
//     PlcTask Outputs/GVL02_IO_EK1101.aOsOutputToEL3702In2[21] <-> Ch1 Sample 21/Ch1 Value
//     PlcTask Outputs/GVL02_IO_EK1101.aOsOutputToEL3702In2[22] <-> Ch1 Sample 22/Ch1 Value
//     PlcTask Outputs/GVL02_IO_EK1101.aOsOutputToEL3702In2[23] <-> Ch1 Sample 23/Ch1 Value
//     PlcTask Outputs/GVL02_IO_EK1101.aOsOutputToEL3702In2[24] <-> Ch1 Sample 24/Ch1 Value
//     PlcTask Outputs/GVL02_IO_EK1101.aOsOutputToEL3702In2[25] <-> Ch1 Sample 25/Ch1 Value
//     PlcTask Outputs/GVL02_IO_EK1101.aOsOutputToEL3702In2[26] <-> Ch1 Sample 26/Ch1 Value
//     PlcTask Outputs/GVL02_IO_EK1101.aOsOutputToEL3702In2[27] <-> Ch1 Sample 27/Ch1 Value
//     PlcTask Outputs/GVL02_IO_EK1101.aOsOutputToEL3702In2[28] <-> Ch1 Sample 28/Ch1 Value
//     PlcTask Outputs/GVL02_IO_EK1101.aOsOutputToEL3702In2[29] <-> Ch1 Sample 29/Ch1 Value
//     PlcTask Outputs/GVL02_IO_EK1101.aOsOutputToEL3702In2[2] <-> Ch1 Sample 2/Ch1 Value
//     PlcTask Outputs/GVL02_IO_EK1101.aOsOutputToEL3702In2[30] <-> Ch1 Sample 30/Ch1 Value
//     PlcTask Outputs/GVL02_IO_EK1101.aOsOutputToEL3702In2[31] <-> Ch1 Sample 31/Ch1 Value
//     PlcTask Outputs/GVL02_IO_EK1101.aOsOutputToEL3702In2[32] <-> Ch1 Sample 32/Ch1 Value
//     PlcTask Outputs/GVL02_IO_EK1101.aOsOutputToEL3702In2[33] <-> Ch1 Sample 33/Ch1 Value
//     PlcTask Outputs/GVL02_IO_EK1101.aOsOutputToEL3702In2[34] <-> Ch1 Sample 34/Ch1 Value
//     PlcTask Outputs/GVL02_IO_EK1101.aOsOutputToEL3702In2[35] <-> Ch1 Sample 35/Ch1 Value
//     PlcTask Outputs/GVL02_IO_EK1101.aOsOutputToEL3702In2[36] <-> Ch1 Sample 36/Ch1 Value
//     PlcTask Outputs/GVL02_IO_EK1101.aOsOutputToEL3702In2[37] <-> Ch1 Sample 37/Ch1 Value
//     PlcTask Outputs/GVL02_IO_EK1101.aOsOutputToEL3702In2[38] <-> Ch1 Sample 38/Ch1 Value
//     PlcTask Outputs/GVL02_IO_EK1101.aOsOutputToEL3702In2[39] <-> Ch1 Sample 39/Ch1 Value
//     PlcTask Outputs/GVL02_IO_EK1101.aOsOutputToEL3702In2[3] <-> Ch1 Sample 3/Ch1 Value
//     PlcTask Outputs/GVL02_IO_EK1101.aOsOutputToEL3702In2[40] <-> Ch1 Sample 40/Ch1 Value
//     PlcTask Outputs/GVL02_IO_EK1101.aOsOutputToEL3702In2[41] <-> Ch1 Sample 41/Ch1 Value
//     PlcTask Outputs/GVL02_IO_EK1101.aOsOutputToEL3702In2[42] <-> Ch1 Sample 42/Ch1 Value
//     PlcTask Outputs/GVL02_IO_EK1101.aOsOutputToEL3702In2[43] <-> Ch1 Sample 43/Ch1 Value
//     PlcTask Outputs/GVL02_IO_EK1101.aOsOutputToEL3702In2[44] <-> Ch1 Sample 44/Ch1 Value
//     PlcTask Outputs/GVL02_IO_EK1101.aOsOutputToEL3702In2[45] <-> Ch1 Sample 45/Ch1 Value
//     PlcTask Outputs/GVL02_IO_EK1101.aOsOutputToEL3702In2[46] <-> Ch1 Sample 46/Ch1 Value
//     PlcTask Outputs/GVL02_IO_EK1101.aOsOutputToEL3702In2[47] <-> Ch1 Sample 47/Ch1 Value
//     PlcTask Outputs/GVL02_IO_EK1101.aOsOutputToEL3702In2[48] <-> Ch1 Sample 48/Ch1 Value
//     PlcTask Outputs/GVL02_IO_EK1101.aOsOutputToEL3702In2[49] <-> Ch1 Sample 49/Ch1 Value
//     PlcTask Outputs/GVL02_IO_EK1101.aOsOutputToEL3702In2[4] <-> Ch1 Sample 4/Ch1 Value
//     PlcTask Outputs/GVL02_IO_EK1101.aOsOutputToEL3702In2[50] <-> Ch1 Sample 50/Ch1 Value
//     PlcTask Outputs/GVL02_IO_EK1101.aOsOutputToEL3702In2[51] <-> Ch1 Sample 51/Ch1 Value
//     PlcTask Outputs/GVL02_IO_EK1101.aOsOutputToEL3702In2[52] <-> Ch1 Sample 52/Ch1 Value
//     PlcTask Outputs/GVL02_IO_EK1101.aOsOutputToEL3702In2[53] <-> Ch1 Sample 53/Ch1 Value
//     PlcTask Outputs/GVL02_IO_EK1101.aOsOutputToEL3702In2[54] <-> Ch1 Sample 54/Ch1 Value
//     PlcTask Outputs/GVL02_IO_EK1101.aOsOutputToEL3702In2[55] <-> Ch1 Sample 55/Ch1 Value
//     PlcTask Outputs/GVL02_IO_EK1101.aOsOutputToEL3702In2[56] <-> Ch1 Sample 56/Ch1 Value
//     PlcTask Outputs/GVL02_IO_EK1101.aOsOutputToEL3702In2[57] <-> Ch1 Sample 57/Ch1 Value
//     PlcTask Outputs/GVL02_IO_EK1101.aOsOutputToEL3702In2[58] <-> Ch1 Sample 58/Ch1 Value
//     PlcTask Outputs/GVL02_IO_EK1101.aOsOutputToEL3702In2[59] <-> Ch1 Sample 59/Ch1 Value
//     PlcTask Outputs/GVL02_IO_EK1101.aOsOutputToEL3702In2[5] <-> Ch1 Sample 5/Ch1 Value
//     PlcTask Outputs/GVL02_IO_EK1101.aOsOutputToEL3702In2[60] <-> Ch1 Sample 60/Ch1 Value
//     PlcTask Outputs/GVL02_IO_EK1101.aOsOutputToEL3702In2[61] <-> Ch1 Sample 61/Ch1 Value
//     PlcTask Outputs/GVL02_IO_EK1101.aOsOutputToEL3702In2[62] <-> Ch1 Sample 62/Ch1 Value
//     PlcTask Outputs/GVL02_IO_EK1101.aOsOutputToEL3702In2[63] <-> Ch1 Sample 63/Ch1 Value
//     PlcTask Outputs/GVL02_IO_EK1101.aOsOutputToEL3702In2[64] <-> Ch1 Sample 64/Ch1 Value
//     PlcTask Outputs/GVL02_IO_EK1101.aOsOutputToEL3702In2[65] <-> Ch1 Sample 65/Ch1 Value
//     PlcTask Outputs/GVL02_IO_EK1101.aOsOutputToEL3702In2[66] <-> Ch1 Sample 66/Ch1 Value
//     PlcTask Outputs/GVL02_IO_EK1101.aOsOutputToEL3702In2[67] <-> Ch1 Sample 67/Ch1 Value
//     PlcTask Outputs/GVL02_IO_EK1101.aOsOutputToEL3702In2[68] <-> Ch1 Sample 68/Ch1 Value
//     PlcTask Outputs/GVL02_IO_EK1101.aOsOutputToEL3702In2[69] <-> Ch1 Sample 69/Ch1 Value
//     PlcTask Outputs/GVL02_IO_EK1101.aOsOutputToEL3702In2[6] <-> Ch1 Sample 6/Ch1 Value
//     PlcTask Outputs/GVL02_IO_EK1101.aOsOutputToEL3702In2[70] <-> Ch1 Sample 70/Ch1 Value
//     PlcTask Outputs/GVL02_IO_EK1101.aOsOutputToEL3702In2[71] <-> Ch1 Sample 71/Ch1 Value
//     PlcTask Outputs/GVL02_IO_EK1101.aOsOutputToEL3702In2[72] <-> Ch1 Sample 72/Ch1 Value
//     PlcTask Outputs/GVL02_IO_EK1101.aOsOutputToEL3702In2[73] <-> Ch1 Sample 73/Ch1 Value
//     PlcTask Outputs/GVL02_IO_EK1101.aOsOutputToEL3702In2[74] <-> Ch1 Sample 74/Ch1 Value
//     PlcTask Outputs/GVL02_IO_EK1101.aOsOutputToEL3702In2[75] <-> Ch1 Sample 75/Ch1 Value
//     PlcTask Outputs/GVL02_IO_EK1101.aOsOutputToEL3702In2[76] <-> Ch1 Sample 76/Ch1 Value
//     PlcTask Outputs/GVL02_IO_EK1101.aOsOutputToEL3702In2[77] <-> Ch1 Sample 77/Ch1 Value
//     PlcTask Outputs/GVL02_IO_EK1101.aOsOutputToEL3702In2[78] <-> Ch1 Sample 78/Ch1 Value
//     PlcTask Outputs/GVL02_IO_EK1101.aOsOutputToEL3702In2[79] <-> Ch1 Sample 79/Ch1 Value
//     PlcTask Outputs/GVL02_IO_EK1101.aOsOutputToEL3702In2[7] <-> Ch1 Sample 7/Ch1 Value
//     PlcTask Outputs/GVL02_IO_EK1101.aOsOutputToEL3702In2[80] <-> Ch1 Sample 80/Ch1 Value
//     PlcTask Outputs/GVL02_IO_EK1101.aOsOutputToEL3702In2[81] <-> Ch1 Sample 81/Ch1 Value
//     PlcTask Outputs/GVL02_IO_EK1101.aOsOutputToEL3702In2[82] <-> Ch1 Sample 82/Ch1 Value
//     PlcTask Outputs/GVL02_IO_EK1101.aOsOutputToEL3702In2[83] <-> Ch1 Sample 83/Ch1 Value
//     PlcTask Outputs/GVL02_IO_EK1101.aOsOutputToEL3702In2[84] <-> Ch1 Sample 84/Ch1 Value
//     PlcTask Outputs/GVL02_IO_EK1101.aOsOutputToEL3702In2[85] <-> Ch1 Sample 85/Ch1 Value
//     PlcTask Outputs/GVL02_IO_EK1101.aOsOutputToEL3702In2[86] <-> Ch1 Sample 86/Ch1 Value
//     PlcTask Outputs/GVL02_IO_EK1101.aOsOutputToEL3702In2[87] <-> Ch1 Sample 87/Ch1 Value
//     PlcTask Outputs/GVL02_IO_EK1101.aOsOutputToEL3702In2[88] <-> Ch1 Sample 88/Ch1 Value
//     PlcTask Outputs/GVL02_IO_EK1101.aOsOutputToEL3702In2[89] <-> Ch1 Sample 89/Ch1 Value
//     PlcTask Outputs/GVL02_IO_EK1101.aOsOutputToEL3702In2[8] <-> Ch1 Sample 8/Ch1 Value
//     PlcTask Outputs/GVL02_IO_EK1101.aOsOutputToEL3702In2[90] <-> Ch1 Sample 90/Ch1 Value
//     PlcTask Outputs/GVL02_IO_EK1101.aOsOutputToEL3702In2[91] <-> Ch1 Sample 91/Ch1 Value
//     PlcTask Outputs/GVL02_IO_EK1101.aOsOutputToEL3702In2[92] <-> Ch1 Sample 92/Ch1 Value
//     PlcTask Outputs/GVL02_IO_EK1101.aOsOutputToEL3702In2[93] <-> Ch1 Sample 93/Ch1 Value
//     PlcTask Outputs/GVL02_IO_EK1101.aOsOutputToEL3702In2[94] <-> Ch1 Sample 94/Ch1 Value
//     PlcTask Outputs/GVL02_IO_EK1101.aOsOutputToEL3702In2[95] <-> Ch1 Sample 95/Ch1 Value
//     PlcTask Outputs/GVL02_IO_EK1101.aOsOutputToEL3702In2[96] <-> Ch1 Sample 96/Ch1 Value
//     PlcTask Outputs/GVL02_IO_EK1101.aOsOutputToEL3702In2[97] <-> Ch1 Sample 97/Ch1 Value
//     PlcTask Outputs/GVL02_IO_EK1101.aOsOutputToEL3702In2[98] <-> Ch1 Sample 98/Ch1 Value
//     PlcTask Outputs/GVL02_IO_EK1101.aOsOutputToEL3702In2[99] <-> Ch1 Sample 99/Ch1 Value
//     PlcTask Outputs/GVL02_IO_EK1101.aOsOutputToEL3702In2[9] <-> Ch1 Sample 9/Ch1 Value
//     PlcTask Outputs/GVL02_IO_EK1101.nEL4732Ch1CycleCount <-> Ch1 CycleCount/Ch1 CycleCount
//   PLC1/PLC1 Instance <-> NC-Task 1 SAF/Axes/Axis 1 Stepper
//     PlcTask Inputs/GVL20_Axis.stAxis1.NcToPlc <-> Outputs/ToPlc
//     PlcTask Outputs/GVL20_Axis.stAxis1.PlcToNc <-> Inputs/FromPlc
//   PLC1/PLC1 Instance <-> NC-Task 1 SAF/Axes/Axis 2 Servo EL
//     PlcTask Inputs/GVL20_Axis.stAxis2.NcToPlc <-> Outputs/ToPlc
//     PlcTask Outputs/GVL20_Axis.stAxis2.PlcToNc <-> Inputs/FromPlc
//   PLC1/PLC1 Instance <-> NC-Task 1 SAF/Axes/Axis 3 Servo A AX
//     PlcTask Inputs/GVL20_Axis.stAxis3.NcToPlc <-> Outputs/ToPlc
//     PlcTask Outputs/GVL20_Axis.stAxis3.PlcToNc <-> Inputs/FromPlc
//   PLC1/PLC1 Instance <-> NC-Task 1 SAF/Axes/Axis 4 Servo B AX
//     PlcTask Inputs/GVL20_Axis.stAxis4.NcToPlc <-> Outputs/ToPlc
//     PlcTask Outputs/GVL20_Axis.stAxis4.PlcToNc <-> Inputs/FromPlc
//   PLC1/PLC1 Instance <-> NC-Task 1 SAF/Axes/Axis 5 Handwheel
//     PlcTask Inputs/GVL20_Axis.stAxis5.NcToPlc <-> Outputs/ToPlc
//     PlcTask Outputs/GVL20_Axis.stAxis5.PlcToNc <-> Inputs/FromPlc
//   PLC1/PLC1 Instance <-> NC-Task 1 SAF/NCI
//     PlcTask Inputs/NCI.in_stItpToPlc <-> Outputs/ToPlc
//     PlcTask Outputs/NCI.out_stPlcToItp <-> Inputs/FromPlc

CONFIGURATION PLC1
    RESOURCE PLC ON TwinCAT3
        TASK extMarkTask(INTERVAL := T#1ms, PRIORITY := 20);
        TASK PlcTask(INTERVAL := T#1ms, PRIORITY := 8);
        TASK PlcTaskFast(INTERVAL := T#100us, PRIORITY := 4);
        PROGRAM extMarksPrg WITH extMarkTask : extMarksPrg;
        PROGRAM MAIN WITH PlcTask : MAIN;
        PROGRAM MAINFast WITH PlcTaskFast : MAINFast;
    END_RESOURCE
END_CONFIGURATION

// ---- DUTs/00_MainBlocks/E_SystemStartupSequence.TcDUT
TYPE E_SystemStartupSequence :
(

	eSystemStart_Start						:= 0,
	eSystemStart_Init						:= 10,
	eSystemStart_LedOn						:= 100,
	eSystemStart_LedOff						,
	eSystemStart_Done						:= 500,
	eSystemStart_ErrorStep 					:= 999,
	eSystemStart_NoError
	
);
END_TYPE
(* End *)

// ---- DUTs/20_Axis/E_AxisReversingSequence.TcDUT
TYPE E_AxisReversingSequence :
(

	eAxisRevSeq_Start						:= 0,
	eAxisRevSeq_Init						:= 10,
	eAxisRevSeq_AxisStartPos1				:= 100,
	eAxisRevSeq_IdleTime1					,
	eAxisRevSeq_AxisStartPos2				,
	eAxisRevSeq_IdleTime2					,
	eAxisRevSeq_AxisStop					,
	eAxisRevSeq_Done						:= 500,
	eAxisRevSeq_ErrorStep 					:= 999,
	eAxisRevSeq_NoError

);
END_TYPE
(* End *)

// ---- DUTs/20_Axis/E_McResetStatus.TcDUT
TYPE E_McResetStatus :
(

	eMcReset_Start							:= 0,
	eMcReset_Init							:= 10,
	eMcReset_ResetHardware					:= 100,
	eMcReset_ResetNc						,
	eMcReset_Done							:= 500,
	eMcReset_ErrorStep 						:= 999,
	eMcReset_NoError

);
END_TYPE
(* End *)

// ---- DUTs/30_EtherCatDiagnostic/E_EcDiacStatus.TcDUT
TYPE E_EcDiacStatus :
(

	eEcDiac_Start							:= 0, 
	eEcDiac_Delay							,
	eEcDiac_ReadMasterState					,
	eEcDiac_ReadSlaveState

);
END_TYPE
(* End *)

// ---- DUTs/30_EtherCatDiagnostic/E_EcGetSlaveName.TcDUT
TYPE E_EcGetSlaveName :
(

	eEcGetSlaveName_Start						:= 0,
	eEcGetSlaveName_Init						:= 10,
	eEcGetSlaveName_ReadAllSlaveAddr			:= 100,
	eEcGetSlaveName_ReadSlaveName				,
	eEcGetSlaveName_Done						:= 500,
	eEcGetSlaveName_ErrorStep 					:= 999,
	eEcGetSlaveName_NoError

);
END_TYPE
(* End *)

// ---- DUTs/30_EtherCatDiagnostic/E_EcSystemStatus.TcDUT
TYPE E_EcSystemStatus :
(

	eEcSystem_Start							:= 0,
	eEcSystem_ReadConfSystem

);
END_TYPE
(* End *)

// ---- DUTs/30_EtherCatDiagnostic/ST_EcTerminalDiagInfo.TcDUT
TYPE ST_EcTerminalDiagInfo :
STRUCT

	nAddr									:UINT;
	sType									:STRING(15);
	sName									:STRING(31);
	sTerminalStatus							:STRING(60);

END_STRUCT
END_TYPE
(* End *)

// ---- DUTs/40_TwinSAFE/ST_AdsAddr.TcDUT
TYPE ST_AdsAddr :
STRUCT

	netId									:AMSNETID;
	port									:WORD;

END_STRUCT
END_TYPE

// ---- DUTs/40_TwinSAFE/TwinSAFE_Connection/AX5805/E_TsDiagnosisObjektsFA10AX5805.TcDUT
TYPE E_TsDiagnosisObjektsFA10AX5805 :
(*******************************************************************************************************
Description			:	Reason for shutdown of CoE objects 0xFA10
Supported terminals : 	AX5805, AX5806
Documentation 		:	AX5805 / AX5806 TwinSAFE drive option cards for the AX5000 servo drive
Version/Date 		:	V1.6.1/15.03.2016
********************************************************************************************************)
(

	eFA10AX5805_NoErrorReaction					:= 16#0000,	(* Error reaction: no error reaction *)
	eFA10AX5805_ErrSafeTorqueOff				:= 16#0040,	(* Error reaction: STO (Safe Torque Off) *)
	eFA10AX5805_ErrSafeStop1					:= 16#0050,	(* Error reaction: SS1 (Safe Stop 1) *)

	eFA10AX5805_StatusWordIncorrect				:= 16#0100,	(* Shutdown reason: The status word was calculated incorrectly *)
	eFA10AX5805_ParametersWrongOrNotLoaded		:= 16#0200,	(* Shutdown reason: The parameters are wrong or not yet loaded *)
	eFA10AX5805_FSOEProtocolWrongState			:= 16#0300,	(* Shutdown reason: FSOE protocol not in state DATA *)
	eFA10AX5805_WrongDriveParameter				:= 16#0400,	(* Shutdown reason: Internal comparison failed. Please check the motor/drive dimensioning/parameterization *)
	eFA10AX5805_ExtCamDetectedUnexpectedly		:= 16#0500,	(* Reason for shutdown position detection: external cam detected unexpectedly *)
	eFA10AX5805_ExtCamRightSideCamWindow		:= 16#0600,	(* Reason for shutdown position detection: external cam detected to the right of the cam window *)
	eFA10AX5805_ExtCamLeftSideCamWindow			:= 16#0700,	(* Reason for shutdown position detection: external cam detected to the left of the cam window *)
	eFA10AX5805_MaxTraversingRangeExceeded		:= 16#0800,	(* Reason for shutdown position detection: the maximum traversing range was exceeded *)
	eFA10AX5805_SS1SwitchedOff					:= 16#5000,	(* Reason for shutdown safety function: The safety function SS1 has switched off *)
	eFA10AX5805_SOSSwitchedOff					:= 16#6800,	(* Reason for shutdown safety function: The safety function SOS has switched off *)
	eFA10AX5805_SSRSwitchedOff					:= 16#8000,	(* Reason for shutdown safety function: The safety function SSR has switched off *)
	eFA10AX5805_SLSSwitchedOff					:= 16#9000,	(* Reason for shutdown safety function: The safety function SLS has switched off *)
	eFA10AX5805_SLPSwitchedOff					:= 16#A000,	(* Reason for shutdown safety function: The safety function SLP has switched off *)
	eFA10AX5805_SMSSwitchedOff					:= 16#A800,	(* Reason for shutdown safety function: The safety function SMS has switched off *)
	eFA10AX5805_SLISwitchedOff					:= 16#B800,	(* Reason for shutdown safety function: The safety function SLI has switched off *)
	eFA10AX5805_SARSwitchedOff					:= 16#C000,	(* Reason for shutdown safety function: The safety function SAR has switched off *)
	eFA10AX5805_SMASwitchedOff					:= 16#C800,	(* Reason for shutdown safety function: The safety function SMA has switched off *)
	eFA10AX5805_SDIpSwitchedOff					:= 16#D000,	(* Reason for shutdown safety function: The safety function SDIp has switched off *)
	eFA10AX5805_SDInSwitchedOff					:= 16#D100	(* Reason for shutdown safety function: The safety function SDIn has switched off *)
	
);
END_TYPE
(* End *)

// ---- DUTs/40_TwinSAFE/TwinSAFE_Connection/AX5805/E_TsErrIndicesFA82AX5805.TcDUT
TYPE E_TsErrIndicesFA82AX5805 :
(*******************************************************************************************************
Description			:	Error indices in CoE objects 0xFA82
Supported terminals : 	AX5805, AX5806
Documentation 		:	AX5805 / AX5806 TwinSAFE drive option cards for the AX5000 servo drive
Version/Date 		:	V1.6.1/15.03.2016
********************************************************************************************************)
(

	eAX5805FA82_NoError									:=	16#0000,	

	eAX5805FA82_FAULT_MAXT_C1							:=	16#0001,	(* The temperature has exceeded the maximum permissible temperature (µC1) *)
	eAX5805FA82_FAULT_MAXT_C2							:=	16#0002,	(* The temperature has exceeded the maximum permissible temperature (µC2) *)
	eAX5805FA82_FAULT_MINT_C1							:=	16#0003,	(* The temperature has fallen below the minimum permissible temperature (µC1) *)
	eAX5805FA82_FAULT_MINT_C2							:=	16#0004,	(* The temperature has fallen below the minimum permissible temperature (µC2) *)

	eAX5805FA82_HW_ERR_MAX_VCC_C1						:=	16#0101,	(* The maximum supply voltage was exceeded (3.3 V) *)
	eAX5805FA82_HW_ERR_MAX_VCC_C2						:=	16#0102,	(* The maximum supply voltage was exceeded (3.3 V) *)
	eAX5805FA82_HW_ERR_MIN_VCC_C1						:=	16#0103,	(* The supply voltage fell below the minimum value (3.3 V) *)
	eAX5805FA82_HW_ERR_MIN_VCC_C2						:=	16#0104,	(* The supply voltage fell below the minimum value (3.3 V) *)

	eAX5805FA82_FAULT_MCTC1_TO							:=	16#0201,	(* The MCTests of µC1 were not carried out completely within the specified time *)
	eAX5805FA82_FAULT_MCTC2_TO							:=	16#0202,	(* The MCTests of µC2 were not carried out completely within the specified time *)
	eAX5805FA82_FAULT_TIMER_C1							:=	16#0203,	(* The global timer was not updated in time *)
	eAX5805FA82_FAULT_TIMER_C2							:=	16#0204,	(* The global timer was not updated in time *)
	eAX5805FA82_FAULT_TS_WDG_TO_C1						:=	16#020C,	(* The TwinSAFE module was not called within the watchdog time *)
	eAX5805FA82_FAULT_TS_WDG_TO_C2						:=	16#020D,	(* The TwinSAFE module was not called within the watchdog time *)
	eAX5805FA82_FAULT_RESET_MC1							:=	16#020E,	(* A reset has occurred in the operation of the controller for µC1. µC2 was not reset thereby *)
	
	eAX5805FA82_FAULT_SERCOMC2							:=	16#0300,	(* An error occurred in the SerComP24C2 module during data transmission *)

	eAX5805FA82_FAULT_SERCOM_1							:=	16#0401,	(* An error occurred in the SerComP24C1 module during data transmission *)
	eAX5805FA82_FAULT_SERCOM_2							:=	16#0402,	(* An error occurred in the SerComP24C1 module during data transmission *)
	eAX5805FA82_FAULT_SERCOM_3							:=	16#0403,	(* An error occurred in the SerComP24C1 module during data transmission *)
	eAX5805FA82_FAULT_SERCOM_4							:=	16#0404,	(* An error occurred in the SerComP24C1 module during data transmission *)
	eAX5805FA82_FAULT_SERCOM_5							:=	16#0405,	(* An error occurred in the SerComP24C1 module during data transmission *)
	eAX5805FA82_FAULT_SERCOM_6							:=	16#0406,	(* An error occurred in the SerComP24C1 module during data transmission *)
	eAX5805FA82_FAULT_SERCOM_7							:=	16#0407,	(* An error occurred in the SerComP24C1 module during data transmission *)
	eAX5805FA82_FAULT_SERCOM_8							:=	16#0408,	(* An error occurred in the SerComP24C1 module during data transmission *)
	eAX5805FA82_FAULT_SERCOM_9							:=	16#0409,	(* An error occurred in the SerComP24C1 module during data transmission *)
	eAX5805FA82_FAULT_SERCOM_A							:=	16#040A,	(* An error occurred in the SerComP24C1 module during data transmission *)
	eAX5805FA82_FAULT_SERCOM_B							:=	16#040B,	(* An error occurred in the SerComP24C1 module during data transmission *)

	eAX5805FA82_FAULT_TEMPSENSOR_1						:=	16#0501,	(* Error in the communication with one of the temperature sensors *)
	eAX5805FA82_FAULT_TEMPSENSOR_2						:=	16#0502,	(* Error in the communication with one of the temperature sensors *)
	eAX5805FA82_FAULT_TEMPSENSOR_3						:=	16#0503,	(* Error in the communication with one of the temperature sensors *)
	eAX5805FA82_FAULT_TEMPSENSOR_4						:=	16#0504,	(* Error in the communication with one of the temperature sensors *)
	eAX5805FA82_FAULT_TEMPSENSOR_5						:=	16#0505,	(* Error in the communication with one of the temperature sensors *)
	eAX5805FA82_FAULT_TEMPSENSOR_6						:=	16#0506,	(* Error in the communication with one of the temperature sensors *)
	eAX5805FA82_FAULT_TEMPSENSOR_7						:=	16#0507,	(* Error in the communication with one of the temperature sensors *)

	eAX5805FA82_FAULT_OUTPUTCOMPARE						:=	16#0601,	(* The values output by µC1 and µC2 differ *)
	eAX5805FA82_FAULT_OUTPUTCOMPAREC2					:=	16#0602,	(* The values output by µC1 and µC2 differ *)

	eAX5805FA82_HW_ERR_MIN_VCC_FPGA						:=	16#0700,	(* The FPGA supply voltage fell below the minimum value (5 V) *)
	eAX5805FA82_HW_ERR_MAX_VCC_FPGA						:=	16#0701,	(* The FPGA supply voltage exceeded the maximum value (5 V) *)

	eAX5805FA82_FAULT_FEEDBACK_C1						:=	16#0710,	(* An error was detected in the feedback channels of µC1 *)
	eAX5805FA82_FAULT_FEEDBACK_C2						:=	16#0711,	(* An error was detected in the feedback channels of µC2 *)

	eAX5805FA82_FAULT_Parameter_C1						:=	16#0720,	(* General parameter error µC1 *)
	eAX5805FA82_FAULT_Parameter_C2						:=	16#0721,	(* General parameter error µC2 *)
	eAX5805FA82_FAULT_Parameter_C1_DRIVE_PROFILE		:=	16#0722,	(* Parameter: unknown parameter index µC1 drive profile *)
	eAX5805FA82_FAULT_Parameter_C1_VENDOR_SPECIFIC		:=	16#0723,	(* Parameter: unknown parameter index µC1 vendor-specific *)
	eAX5805FA82_FAULT_Parameter_C2_DRIVE_PROFILE		:=	16#0724,	(* Parameter: unknown parameter index µC2 drive profile *)
	eAX5805FA82_FAULT_Parameter_C2_VENDOR_SPECIFIC		:=	16#0725,	(* Parameter: unknown parameter index µC2 vendor-specific *)
	eAX5805FA82_FAULT_PDO_MAPPING_FSOE_COMMAND			:=	16#0726,	(* PDO mapping axis 1/2: FSOE COMMAND error *)
	eAX5805FA82_FAULT_PDO_MAPPING_LENGTH				:=	16#0727,	(* PDO mapping axis 1: Length_Error *)
	eAX5805FA82_FAULT_PDO_MAPPING_STO_K1				:=	16#0728,	(* PDO mapping axis 1: STO error *)
	eAX5805FA82_FAULT_PDO_MAPPING_SS1_1_K1				:=	16#0729,	(* PDO mapping axis 1: Error SS1_1 *)
	eAX5805FA82_FAULT_PDO_MAPPING_SS2_1_K1				:=	16#072A,	(* PDO mapping axis 1: Error SS2_1 *)
	eAX5805FA82_FAULT_PDO_MAPPING_SOS_1_K1				:=	16#072B,	(* PDO mapping axis 1: SS2_1 error *)
	eAX5805FA82_FAULT_PDO_MAPPING_SSR_1_K1				:=	16#072C,	(* PDO mapping axis 1: SSR_1 error *)
	eAX5805FA82_FAULT_PDO_MAPPING_SDIp_K1				:=	16#072D,	(* PDO mapping axis 1: SDIp error *)
	eAX5805FA82_FAULT_PDO_MAPPING_SDIn_K1				:=	16#072E,	(* PDO mapping axis 1: SDIn error *)
	eAX5805FA82_FAULT_PDO_MAPPING_Error_ACK_K1			:=	16#072F,	(* PDO mapping axis 1: Error_ACK error *)
	
	eAX5805FA82_FAULT_PDO_MAPPING_Error_CRC0			:=	16#0730,	(* PDO mapping axis 1/2: FSOE CRC0 error *)
	eAX5805FA82_FAULT_PDO_MAPPING_STO_K2				:=	16#0731,	(* PDO mapping axis 2: STO error *)
	eAX5805FA82_FAULT_PDO_MAPPING_SS1_1_K2				:=	16#0732,	(* PDO mapping axis 2: Error SS1_1 *)
	eAX5805FA82_FAULT_PDO_MAPPING_SS2_1_K2				:=	16#0733,	(* PDO mapping axis 2: Error SS2_1 *)
	eAX5805FA82_FAULT_PDO_MAPPING_SOS_1_K2				:=	16#0734,	(* PDO mapping axis 2: SS2_1 error *)
	eAX5805FA82_FAULT_PDO_MAPPING_SSR_1_K2				:=	16#0735,	(* PDO mapping axis 2: SSR_1 error *)
	eAX5805FA82_FAULT_PDO_MAPPING_SDIp_K2				:=	16#0736,	(* PDO mapping axis 2: SDIp error *)
	eAX5805FA82_FAULT_PDO_MAPPING_SDIn_K2				:=	16#0737,	(* PDO mapping axis 2: SDIn error *)
	eAX5805FA82_FAULT_PDO_MAPPING_Error_ACK_K2			:=	16#0738,	(* PDO mapping axis 2: Error_ACK error *)
	eAX5805FA82_FAULT_PDO_MAPPING_Error_CRC1			:=	16#0739,	(* PDO mapping axis 2: FSOE CRC1 error *)
	eAX5805FA82_FAULT_PDO_MAPPING_Error_ConnID			:=	16#073A,	(* PDO mapping axis 1/2: FSOE ConnID error *)
	eAX5805FA82_FAULT_PDO_MAPPING_SSM_1_K1				:=	16#073B,	(* PDO mapping axis 1: SSM_1_K1 error *)
	eAX5805FA82_FAULT_PDO_MAPPING_SSM_1_K2				:=	16#073C,	(* PDO mapping axis 2: SSM_1_K2 error *)
	eAX5805FA82_FAULT_PDO_MAPPING_SSM_2_K1				:=	16#073D,	(* PDO mapping axis 1: SSM_2_K1 error *)
	eAX5805FA82_FAULT_PDO_MAPPING_SSM_2_K2				:=	16#073E,	(* PDO mapping axis 2: SSM_2_K2 error *)	

	eAX5805FA82_FAULT_WRONG_MOTORCONSTRUCTIONTYPE_K1	:=	16#0740,	(* Register communication: parameterized motor type for axis 1 does not correspond to the connected motor *)
	eAX5805FA82_FAULT_UNKNOWN_MOTOR_TYPE_K1				:=	16#0741,	(* Register communication: parameterized motor type for axis 1 is unknown *)
	eAX5805FA82_FAULT_WRONG_MOTORCONSTRUCTIONTYPE_K2	:=	16#0742,	(* Register communication: parameterized motor type for axis 2 does not correspond to the connected motor *)
	eAX5805FA82_FAULT_UNKNOWN_MOTOR_TYPE_K2				:=	16#0743,	(* Register communication: parameterized motor type for axis 2 is unknown *)
	eAX5805FA82_FAULT_NUM_OF_POLEPAIRS_K1				:=	16#0744,	(* Register communication: parameterized number of pole pairs for axis 1 does not correspond to the connected motor *)
	eAX5805FA82_FAULT_NUM_OF_POLEPAIRS_K2				:=	16#0745,	(* Register communication: parameterized number of pole pairs for axis 2 does not correspond to the connected motor *)
	eAX5805FA82_FAULT_WRONG_MOTOR_CONFIGURED_K1			:=	16#0746,	(* Register communication: parameterized motor type for axis 1 does not correspond to the connected motor *)
	eAX5805FA82_FAULT_WRONG_MOTOR_CONFIGURED_K2			:=	16#0747,	(* Register communication: parameterized motor type for axis 2 does not correspond to the connected motor *)
	eAX5805FA82_FAULT_RXPDO_LENGTH						:=	16#0748,	(* PDO mapping: RXPDO length is wrong *)
	eAX5805FA82_FAULT_TXPDO_LENGTH						:=	16#0749,	(* PDO mapping: TXPDO length is wrong *)
	eAX5805FA82_FAULT_UNKNOWN_RXPDO_INDEX				:=	16#074A,	(* PDO mapping: RXPDO index is unknown *)
	eAX5805FA82_FAULT_UNKNOWN_TXPDO_INDEX				:=	16#074B,	(* PDO mapping: TXPDO index is unknown *)
	eAX5805FA82_FAULT_WRONG_NUMBER_OF_AXLE				:=	16#074C, 	(* The parameterized number of axes does not correspond to the number detected *)

	eAX5805FA82_FAULT_CRC_INIT_C1						:=	16#1001,	(* An incorrect checksum at µC1 was determined during PowerOn reset *)
	eAX5805FA82_FAULT_CRC_INIT_C2						:=	16#1002,	(* An incorrect checksum at µC2 was determined during PowerOn reset *)
	eAX5805FA82_FAULT_CRC_C1							:=	16#1003,	(* An incorrect checksum was determined for µC1 during operation *)
	eAX5805FA82_FAULT_CRC_C2							:=	16#1004,	(* An incorrect checksum was determined for µC2 during operation *)
	eAX5805FA82_FAULT_RAM_C1							:=	16#1011,	(* An error occurred during the RAM test of µC1 - Typical error reaction time (125µs) *)
	eAX5805FA82_FAULT_RAM_C2							:=	16#1012,	(* An error occurred during the RAM test of µC2 - Typical error reaction time (125µs) *)
	eAX5805FA82_FAULT_RAM_CHECKERBOARD_C1				:=	16#1013,	(* An error occurred during the RAM test of µC1 *)
	eAX5805FA82_FAULT_RAM_CHECKERBOARD_C2				:=	16#1014,	(* An error occurred during the RAM test of µC2 *)
	eAX5805FA82_FAULT_GLBL_TMR							:=	16#1021,	(* The global timer is not working correctly - Typical error reaction time (125µs) *)
	eAX5805FA82_FAULT_SPLIM1							:=	16#1031,	(* Stack overruns are no longer being intercepted correctly *)
	eAX5805FA82_FAULT_SPLIM2							:=	16#1032,	(* Stack overruns are no longer being intercepted correctly *)

	eAX5805FA82_FAULT_OPCT_GRP_C1						:=	16#1100,	(* The opcode test for µC1 has failed *)

	eAX5805FA82_FAULT_OPCT_GRP_C2						:=	16#1300,	(* The opcode test for µC2 has failed *)

	eAX5805FA82_FAULT_ESS_CRC_C1						:=	16#1801,	(* Different check sums were determined in the TwinSAFE telegrams *)
	eAX5805FA82_FAULT_ESS_CRC_C2						:=	16#1802,	(* Different check sums were determined in the TwinSAFE telegrams *)
	eAX5805FA82_FAULT_SW_MAIN1_C1						:=	16#1803,	(* The default case of the main loop of µC1 was called *)
	eAX5805FA82_FAULT_SW_MAIN1_C2						:=	16#1804,	(* The default case of the main loop of µC2 was called *)
	eAX5805FA82_FAULT_ESLCONID_PRJCRCRD					:=	16#1805,	(* The Connection ID is not zero when reading the project CRC *)
	eAX5805FA82_FAULT_ESLCONID_PRJCRCWR					:=	16#1806,	(* The Connection ID is not zero when writing the project CRC *)
	eAX5805FA82_FAULT_SIZE_EEVONDOR_EXID				:=	16#1807,	(* An address was accessed that lies outside the vendor range in the EEPROM *)

	eAX5805FA82_FAULT_COM_C1C2							:=	16#5100,	(* Communication between µC1 and µC2 is disturbed *)
	eAX5805FA82_FAULT_ISR_SNT_FEEDBACK					:=	16#5101,	(* High priority ISR: communication interrupted: switched mode power supply feedback - Typical error reaction time (125µs) *)
	eAX5805FA82_FAULT_ISR_ANGLE_K1						:=	16#5102,	(* High priority ISR: communication interrupted: axis 1 angle - Typical error reaction time (125µs) *)
	eAX5805FA82_FAULT_ISR_ANGLE_K2						:=	16#5103,	(* High priority ISR: communication interrupted: axis 2 angle - Typical error reaction time (125µs) *)
	eAX5805FA82_FAULT_ISR_DELTA_K1						:=	16#5104,	(* High priority ISR: communication interrupted: axis 1 distance travelled - Typical error reaction time (125µs) *)
	eAX5805FA82_FAULT_ISR_DELTA_K2						:=	16#5105,	(* High priority ISR: communication interrupted: axis 2 distance travelled - Typical error reaction time (125µs) *)
	eAX5805FA82_FAULT_ISR_VELO_K1						:=	16#5106,	(* High priority ISR: communication interrupted: axis 1 velocity - Typical error reaction time (125µs) *)
	eAX5805FA82_FAULT_ISR_VELO_K2						:=	16#5107,	(* High priority ISR: communication interrupted: axis 2 velocity - Typical error reaction time (125µs) *)
	eAX5805FA82_FAULT_ISR_TEST_FEEDBACK					:=	16#5108,	(* High priority ISR: communication interrupted: feedback from switch-off channels - Typical error reaction time (125µs) *)
	eAX5805FA82_FAULT_TIMEOUT_REG_AX5000_CONTROL		:=	16#5109,	(* Register communication: AX5000 does not answer in time: Controlword *)
	eAX5805FA82_FAULT_TIMEOUT_REG_AX5000_STATUS			:=	16#510A,	(* Register communication: AX5000 does not answer in time: Statusword *)
	eAX5805FA82_FAULT_TIMEOUT_REG_AX5000_REGADR			:=	16#510B,	(* Register communication: AX5000 does not answer in time: Register address *)
	eAX5805FA82_FAULT_TIMEOUT_REG_AX5000_REGDATA		:=	16#510C,	(* Register communication: AX5000 does not answer in time: Register data *)
	eAX5805FA82_FAULT_TIMEOUT_REG_AX5000_CRC			:=	16#510D,	(* Register communication: AX5000 does not answer in time: CRC *)
	eAX5805FA82_FAULT_UNKNOWN_AX5000_INTERFACE			:=	16#510E,	(* Register communication: unknown interface to the AX5000 *)
	eAX5805FA82_FAULT_COMERROR_AX5000_INTERFACE			:=	16#510F,	(* Register communication: the interface to the AX5000 has a communication error *)
	eAX5805FA82_FAULT_WRITE_HW_VERSION_AX5805_0			:=	16#5110,	(* Values could not be written to the register in the AX5000 *)
	eAX5805FA82_FAULT_WRITE_HW_VERSION_AX5805_1			:=	16#5111,	(* Values could not be written to the register in the AX5000 *)
	eAX5805FA82_FAULT_WRITE_HW_VERSION_AX5805_2			:=	16#5112,	(* Values could not be written to the register in the AX5000 *)
	eAX5805FA82_FAULT_WRITE_HW_VERSION_AX5805_3			:=	16#5113,	(* Values could not be written to the register in the AX5000 *)
	eAX5805FA82_FAULT_EXT_ADC_ADDRESS					:=	16#5114,	(* High priority ISR: External ADC: an impermissible address was read *)
	eAX5805FA82_FAULT_REGISTER_AX5000_CRC_ERROR			:=	16#5115,	(* Register communication with the AX5000: telegram has a CRC error *)
	eAX5805FA82_FAULT_CYCLIC_AX5000_CRC_ERROR			:=	16#5116,	(* High priority ISR: cyclic communication with the AX5000: telegram has a CRC error - Typical error reaction time (125µs) *)
	eAX5805FA82_FAULT_UNKNOWN_REGISTER_ADDRESS			:=	16#5117,	(* Register communication: Addressed register is unknown *)
	eAX5805FA82_FAULT_AX5000_NOT_READY					:=	16#5118,	(* High priority ISR: cyclic communication with the AX5000: AX5000 signals a communication error - Typical error reaction time (125µs) *)
	eAX5805FA82_FAULT_C1C2_SYNC_LOST					:=	16#5119,	(* High priority ISR: cyclic communication between µC1 and µC2: Communication error - Typical error reaction time (125µs) *)

	eAX5805FA82_FAULT_SET_MAPPED_STATE					:=	16#5C00,	(* Mapped safety functions: error while setting the state *)
	eAX5805FA82_FAULT_RESET_MAPPED_STATE				:=	16#5C01,	(* Mapped safety functions: error while resetting the state *)
	eAX5805FA82_FAULT_MAPPED_FUNCTION					:=	16#5C02,	(* Mapped safety functions: invalid mapping, function does not exist *)
	eAX5805FA82_FAULT_MAPPED_INSTANCE					:=	16#5C03,	(* Mapped safety functions: invalid mapping, instance does not exist *)

	eAX5805FA82_FAULT_STO_MODE							:=	16#5E02,	(* The requested STO mode is invalid *)
	eAX5805FA82_FAULT_SDI_MODE							:=	16#5E03,	(* The requested SDI mode is invalid *)
	eAX5805FA82_FAULT_UNDEFINED_ERRORREACTION			:=	16#5E04,	(* Error reaction: invalid error reaction, error reaction does not exist *)

	eAX5805FA82_FAULT_CRC_COMPARE_C1					:=	16#5F00,	(* Incorrect checksum detected during comparison by µC1 *)
	eAX5805FA82_FAULT_CRC_COMPARE_C2					:=	16#5F01,	(* Incorrect checksum detected during comparison by µC2 *)
	eAX5805FA82_FAULT_TMR2_INTERRUPT_C1					:=	16#5F02,	(* MC_Test: Timer2 has triggered an interrupt on µC1. HighPrioISR was not called in time *)
	eAX5805FA82_FAULT_TMR2_INTERRUPT_C2					:=	16#5F03,	(* MC_Test: Timer2 has triggered an interrupt on µC2. HighPrioISR was not called in time *)
	eAX5805FA82_FAULT_SWITCHOFF_TEST					:=	16#5F04,	(* MC_Test: the test of the switch-off channels has failed *)
	eAX5805FA82_FAULT_NO_SYNC							:=	16#5F05,	(* No SYNC signal *)
	eAX5805FA82_FAULT_UNKNOWN_AXLE						:=	16#5F06,	(* The requested axis is unknown *)
	eAX5805FA82_FAULT_FPGA_C2							:=	16#5F07,	(* The status of the FPGA is incorrect *)
	eAX5805FA82_FAULT_ANGLE_FORMAT_C1					:=	16#5F08,	(* The angles OF µC1 read-in have the wrong format - Typical error reaction TIME (125µS) *)
	eAX5805FA82_FAULT_ANGLE_FORMAT_C2					:=	16#5F09,	(* The angles of µC2 read-in have the wrong format - Typical error reaction time (125µs) *)
	eAX5805FA82_FAULT_SAFE_MAIN_STATE					:=	16#5F0A,	(* Unknown state requested *)
	eAX5805FA82_FAULT_STARTUP_FAILED					:=	16#5F0B,	(* Error during start-up *)
	eAX5805FA82_FAULT_MOTION_DETECTION					:=	16#5F0C,	(* Motion detection error - Typical error reaction time (125µs) *)

	eAX5805FA82_FAULT_PARAMETER_FSOE_VENDOR_ID			:=	16#6000,	(* Incorrect vendor ID transmitted *)
	eAX5805FA82_FAULT_PARAMETER_FSOE_MODULE_IDENT		:=	16#6001,	(* Incorrect module ID transmitted *)
	eAX5805FA82_FAULT_PARAMETER_FSOE_CRC				:=	16#6002		(* CRC of the AX5805 parameters does not match the transmitted CRC (please check parameters; if necessary, activate System Manager configuration and reload safety project into the EL69xx) *)
);
END_TYPE
(* End *)

// ---- DUTs/40_TwinSAFE/TwinSAFE_Connection/AX5805/ST_TsControlWordAX5805.TcDUT
TYPE ST_TsControlWordAX5805 :
(*******************************************************************************************************
Description			:	Standard control Word of AX5805/6 terminal
Supported terminals : 	AX5805, AX5806
Documentation 		:	AX5805 / AX5806 TwinSAFE drive option cards for the AX5000 servo drive
Version/Date 		:	V1.6.1/15.03.2016
********************************************************************************************************)
STRUCT
	
	bSafeTorqueOff_STO 						:BOOL;
	bSafeStop1_SS1_1 						:BOOL;
	bSafeStop2_SS2_1 						:BOOL;
	bSafeOperatingStop_SOS_1 				:BOOL;
	bSafeSpeedRange_SSR_1 					:BOOL;
	bSafeDirectionPositive_SDIp				:BOOL;
	bSafeDirectionNegative_SDIn				:BOOL;
	bErrorAcknowledge_ErrAck				:BOOL;
	bNotInUseBit8	 						:BOOL;
	bNotInUseBit9	 						:BOOL;
	bNotInUseBit10	 						:BOOL;
	bNotInUseBit11	 						:BOOL;
	bNotInUseBit12	 						:BOOL;
	bNotInUseBit13	 						:BOOL;
	bNotInUseBit14	 						:BOOL;
	bNotInUseBit15				 			:BOOL;
	
END_STRUCT
END_TYPE
(* End *)

// ---- DUTs/40_TwinSAFE/TwinSAFE_Connection/AX5805/ST_TsDiagObjectsFA10AX5805.TcDUT
TYPE ST_TsDiagObjectsFA10AX5805 :
(*******************************************************************************************************
Description			:	Reason for shutdown of CoE objects 0xFA10
Supported terminals : 	AX5805, AX5806
Documentation 		:	AX5805 / AX5806 TwinSAFE drive option cards for the AX5000 servo drive
Version/Date 		:	V1.6.1/15.03.2016
********************************************************************************************************)
STRUCT

	nDummyData1								:ARRAY[0..3] OF UINT;
	nSoftwareCrcC1							:UINT;
	nSoftwareCrcC2							:UINT;
	nReasonForShutdownAxis1					:UINT;
	nReasonForShutdownAxis2					:UINT;
	
END_STRUCT
END_TYPE
(* End *)

// ---- DUTs/40_TwinSAFE/TwinSAFE_Connection/AX5805/ST_TsErrIndicesFA82AX5805.TcDUT
TYPE ST_TsErrIndicesFA82AX5805 :
(*******************************************************************************************************
Description			:	Error indices in CoE objects 0xFA82
Supported terminals : 	AX5805, AX5806
Documentation 		:	AX5805 / AX5806 TwinSAFE drive option cards for the AX5000 servo drive
Version/Date 		:	V1.6.1/15.03.2016
********************************************************************************************************)
STRUCT

(* Diagnosis motion contoler 1/2 *)
	nDiagnosisMC1							:UINT;
	nDiagnosisMC2							:UINT;

(* Error motion contoler 1/2 *)
	nErrorMC1								:UINT;
	nErrorMC2								:UINT;

END_STRUCT
END_TYPE
(* End *)

// ---- DUTs/40_TwinSAFE/TwinSAFE_Connection/AX5805/ST_TsStatusWordAX5805.TcDUT
TYPE ST_TsStatusWordAX5805 :
(*******************************************************************************************************
Description			:	Standard status Word of AX5805/6 terminal
Supported terminals : 	AX5805, AX5806
Documentation 		:	AX5805 / AX5806 TwinSAFE drive option cards for the AX5000 servo drive
Version/Date 		:	V1.6.1/15.03.2016
********************************************************************************************************)
STRUCT
	
	bSafeTorqueOff_STO 						:BOOL;
	bSafeSpeedMonitor_SSM_1					:BOOL;
	bSafeSpeedMonitor_SSM_2					:BOOL;
	bSafeOperatingStop_SOS_1 				:BOOL;
	bSafeSpeedRange_SSR_1 					:BOOL;
	bSafeDirectionPositive_SDIp				:BOOL;
	bSafeDirectionNegative_SDIn				:BOOL;
	bErrorAcknowledge_ErrAck				:BOOL;
	bNotInUseBit8	 						:BOOL;
	bNotInUseBit9	 						:BOOL;
	bNotInUseBit10	 						:BOOL;
	bNotInUseBit11	 						:BOOL;
	bNotInUseBit12	 						:BOOL;
	bNotInUseBit13	 						:BOOL;
	bNotInUseBit14	 						:BOOL;
	bNotInUseBit15	 						:BOOL;

END_STRUCT
END_TYPE
(* End *)

// ---- DUTs/40_TwinSAFE/TwinSAFE_Connection/EK1914/ST_TsDiagObjectsBitsEK1914.TcDUT
TYPE ST_TsDiagObjectsBitsEK1914 :
(*******************************************************************************************************
Description			:	Index 16#800E Diagnostic objects
Supported terminals : 	EK1914
Documentation 		:	EK1914 TwinSAFE input/output terminal with 2 fail-safe inputs and 2 fail-safe outputs
Version/Date 		:	V1.2.0/08.03.2016
********************************************************************************************************)
STRUCT

(* Sensor test error *)
	bErrInput1								:BOOL;	(* Error input 1 - Bit0 - Error at input 1 *)
	bErrInput2								:BOOL;	(* Error input 2 - Bit1 - Error at input 2 *)

(* Error during two channel evaluation *)
	bErrFirstInputPair						:BOOL;	(* Error input 1..2 - Bit0 - Error in the first input pair *)

(* Error in the safety mat operating mode: input pair disagree *)
	bMatOpModeErrFirstInputPair				:BOOL;	(* Error input 1..2 - Bit1, Bit0 - Mat operating mode - Error in the first input pair *)

(* Error in the safety mat operating mode: external supply *)
	bMatOpModeExtSupplyErrInput1			:BOOL;	(* Error input 1 - Bit0 - Mat operating mode external supply - Error at input 1 *)
	bMatOpModeExtSupplyErrInput2			:BOOL;	(* Error input 2 - Bit1 - Mat operating mode external supply - Error at input 2 *)

(* Diagnosis μC1 *)
	bCcErrOutput1							:BOOL;	(* Diagnosis μC1 - Value  5    - Cross-circuit output 1 and output 2 *)
	bCcErrOutput2							:BOOL;	(* Diagnosis μC1 - Value  6    - Cross-circuit output 1 and output 2 *)
	bOvervoltage							:BOOL;	(* Diagnosis μC1 - Value 10    - Overvoltage *)
	bUndervoltage							:BOOL;	(* Diagnosis μC1 - Value 11    - Undervoltage *)
	bErrTestFieldVolSitches					:BOOL;	(* Diagnosis μC1 - Value 21-27 - Error when testing the field voltage switches *)
	bErrStartUpOutputCircuit				:BOOL;	(* Diagnosis μC1 - Value 30-33 - Start-up of the output circuit failed *)

	bExtSupply0VOutput1MicroC1				:BOOL;	(* Diagnosis μC1 - Value 101   - External supply 0 V output 1, detected with set output *)
	bExtSupply24VOutput1MicroC1				:BOOL;	(* Diagnosis μC1 - Value 102   - External supply 24 V output 1 *)
	bExtSupply0VOutput2MicroC1				:BOOL;	(* Diagnosis μC1 - Value 103   - External supply 0 V output 2, detected with set output *)
	bExtSupply24VOutput2MicroC1				:BOOL;	(* Diagnosis μC1 - Value 104   - External supply 24 V output 2 *)

(* Diagnosis μC2 *)
	bExtSupply0VOutput1MicroC2				:BOOL;	(* Diagnosis μC2 - Value 201 - External supply 0 V output 1, detected with set output *)
	bExtSupply24VOutput1MicroC2				:BOOL;	(* Diagnosis μC2 - Value 202 - External supply 24 V output 1 *)
	bExtSupply0VOutput2MicroC2				:BOOL;	(* Diagnosis μC2 - Value 203 - External supply 0 V output 2, detected with set output *)
	bExtSupply24VOutput2MicroC2				:BOOL;	(* Diagnosis μC2 - Value 204 - External supply 24 V output 2 *)
	
END_STRUCT
END_TYPE
(* End *)

// ---- DUTs/40_TwinSAFE/TwinSAFE_Connection/EK1914/ST_TsDiagObjectsEK1914.TcDUT
TYPE ST_TsDiagObjectsEK1914 :
(*******************************************************************************************************
Description			:	Index 16#800E Diagnostic objects
Supported terminals : 	EK1914
Documentation 		:	EK1914 TwinSAFE input/output terminal with 2 fail-safe inputs and 2 fail-safe outputs
Version/Date 		:	V1.2.0/08.03.2016
********************************************************************************************************)
STRUCT
	
	nDummyData1								:ARRAY[0..8] OF UINT;

(* Sensor test error *)
	nSensorTestError						:UINT;

(* Error during two channel evaluation *)
	nDuringTwoChannelEvaluationError		:UINT;

(* Error in the safety mat operating mode: input pair disagree *)
	nMatModeInputPairDisagreeError			:UINT;

(* Error in the safety mat operating mode: external supply *)
	nMatModeExternalSupplyError				:UINT;

(* Diagnosis μC1 *)
	nDiagnosisMicroC1						:UINT;

(* Diagnosis μC2 *)
	nDiagnosisMicroC2						:UINT;

	nDummyData2								:ARRAY[0..48] OF UINT;

END_STRUCT
END_TYPE
(* End *)

// ---- DUTs/40_TwinSAFE/TwinSAFE_Connection/EL1904/ST_TsDiagObjectsBitsEL1904.TcDUT
TYPE ST_TsDiagObjectsBitsEL1904 :
(*******************************************************************************************************
Description			:	Index 16#800E Diagnostic objects
Supported terminals : 	EL1904
Documentation 		:	EL1904 TwinSAFE input terminal with 4 fail-safe inputs
Version/Date 		:	V1.5.2/02.10.2015
********************************************************************************************************)
STRUCT
	
(* Sensor test error *)
	bErrInput1								:BOOL;	(* Error input 1 - Bit0 - Error at input 1 *)
	bErrInput2								:BOOL;	(* Error input 2 - Bit1 - Error at input 2 *)
	bErrInput3								:BOOL;	(* Error input 3 - Bit2 - Error at input 3 *)
	bErrInput4								:BOOL;	(* Error input 4 - Bit3 - Error at input 4 *)

(* Error during two channel evaluation *)
	bErrFirstInputPair						:BOOL;	(* Error input 1..2 - Bit0 - Error in the first input pair *)
	bErrSecondInputPair						:BOOL;	(* Error input 3..4 - Bit1 - Error in the second input pair *)

(* Error in the safety mat operating mode: input pair disagree *)
	bMatOpModeErrFirstInputPair				:BOOL;	(* Error input 1..2 - Bit1, Bit0 - Mat operating mode - Error in the first input pair *)
	bMatOpModeErrSecondInputPair			:BOOL;	(* Error input 3..4 - Bit3, Bit2 - Mat operating mode - Error in the second input pair *)

(* Error in the safety mat operating mode: external supply *)
	bMatOpModeExtSupplyErrInput1			:BOOL;	(* Error input 1 - Bit0 - Mat operating mode external supply - Error at input 1 *)
	bMatOpModeExtSupplyErrInput2			:BOOL;	(* Error input 2 - Bit1 - Mat operating mode external supply - Error at input 2 *)
	bMatOpModeExtSupplyErrInput3			:BOOL;	(* Error input 3 - Bit2 - Mat operating mode external supply - Error at input 3 *)
	bMatOpModeExtSupplyErrInput4			:BOOL;	(* Error input 4 - Bit3 - Mat operating mode external supply - Error at input 4 *)
	
END_STRUCT
END_TYPE
(* End *)

// ---- DUTs/40_TwinSAFE/TwinSAFE_Connection/EL1904/ST_TsDiagObjectsEL1904.TcDUT
TYPE ST_TsDiagObjectsEL1904 :
(*******************************************************************************************************
Description			:	Index 16#800E Diagnostic objects
Supported terminals : 	EL1904
Documentation 		:	EL1904 TwinSAFE input terminal with 4 fail-safe inputs
Version/Date 		:	V1.5.2/02.10.2015
********************************************************************************************************)
STRUCT

	nDummyData1								:ARRAY[0..8] OF UINT;

(* Sensor test error *)
	nSensorTestError						:UINT;

(* Error during two channel evaluation *)
	nDuringTwoChannelEvaluationError		:UINT;

(* Error in the safety mat operating mode: input pair disagree *)
	nMatModeInputPairDisagreeError			:UINT;

(* Error in the safety mat operating mode: external supply *)
	nMatModeExternalSupplyError				:UINT;

	nDummyData2								:ARRAY[0..2] OF UINT;

END_STRUCT
END_TYPE
(* End *)

// ---- DUTs/40_TwinSAFE/TwinSAFE_Connection/EL2904/ST_TsDiagObjectsBitsEL2904.TcDUT
TYPE ST_TsDiagObjectsBitsEL2904 :
(*******************************************************************************************************
Description			:	Index 16#800E Diagnostic objects
Supported terminals : 	EL2904
Documentation 		:	EL2904 TwinSAFE output terminal with 4 fail-safe outputs
Version/Date 		:	V1.6.2/02.10.2015
********************************************************************************************************)
STRUCT
	
(* Error at the outputs *)
	bEsOrCcErrOutput1						:BOOL;	(* Error output 1 - Bit0 - External supply or cross circuit *)
	bEsOrCcErrOutput2						:BOOL;	(* Error output 2 - Bit1 - External supply or cross circuit *)
	bEsOrCcErrOutput3						:BOOL;	(* Error output 3 - Bit2 - External supply or cross circuit *)
	bEsOrCcErrOutput4						:BOOL;	(* Error output 4 - Bit3 - External supply or cross circuit *)
	bOlOrCvErrOutput1						:BOOL;	(* Error output 1 - Bit4 - Open load or current below minimum value of 20 mA or current above maximum value of 500mA *)
	bOlOrCvErrOutput2						:BOOL;	(* Error output 2 - Bit5 - Open load or current below minimum value of 20 mA or current above maximum value of 500mA *)
	bOlOrCvErrOutput3						:BOOL;	(* Error output 3 - Bit6 - Open load or current below minimum value of 20 mA or current above maximum value of 500mA *)
	bOlOrCvErrOutput4						:BOOL;	(* Error output 4 - Bit7 - Open load or current below minimum value of 20 mA or current above maximum value of 500mA *)

(* Supply error *)
	bFieldVoltageTooHigh					:BOOL;	(* Supply error - Bit 0 - Field voltage too high *)
	bFieldVoltageTooLow						:BOOL;	(* Supply error - Bit 1 - Field voltage too low *)

(* Temperature error *)
	nOvertemperatureC1						:BOOL;	(* Temperature error - Bit 0 - Overtemperature µC1 *)
	nOvertemperatureC2						:BOOL;	(* Temperature error - Bit 1 - Overtemperature µC2 *)
	nOvertemperatureOutputs					:BOOL;	(* Temperature error - Bit 2 - Overtemperature of the output board *)
	nTemperatureTooLowC1					:BOOL;	(* Temperature error - Bit 3 - Temperature too low µC1 *)
	nTemperatureTooLowC2					:BOOL;	(* Temperature error - Bit 4 - Temperature too low µC2 *)
	nTemperatureTooLowOutputs				:BOOL;	(* Temperature error - Bit 5 - Temperature of the output board too low *)
	nOvertemperatureDiffBoard				:BOOL;	(* Temperature error - Bit 6 - Temperature difference on the processor board too large *)
	nOvertemperatureDiffBetwBoards			:BOOL;	(* Temperature error - Bit 7 - Temperature difference between the boards is too large *)
	
END_STRUCT
END_TYPE
(* End *)

// ---- DUTs/40_TwinSAFE/TwinSAFE_Connection/EL2904/ST_TsDiagObjectsEL2904.TcDUT
TYPE ST_TsDiagObjectsEL2904 :
(*******************************************************************************************************
Description			:	Index 16#800E Diagnostic objects
Supported terminals : 	EL2904
Documentation 		:	EL2904 TwinSAFE output terminal with 4 fail-safe outputs
Version/Date 		:	V1.6.2/02.10.2015
********************************************************************************************************)
STRUCT
	
	nDummyData1								:ARRAY[0..10] OF UINT;

(* Error at the outputs *)
	nErrorOutputs							:UINT;

(* Supply error *)
	nSupplyError							:UINT;

(* Temperature error *)
	nTemperatureError						:UINT;

	nDummyData2								:ARRAY[0..1] OF UINT;

END_STRUCT
END_TYPE
(* End *)

// ---- DUTs/40_TwinSAFE/TwinSAFE_Connection/E_TsCycleDiagObj.TcDUT
TYPE E_TsCycleDiagObj :
(*******************************************************************************************************
Description			:	Enumeration read diagnosis objects steps 
Supported terminals : 	EL1904, EL2904, AX5805, AX5806
Date 				:	04.04.2016
********************************************************************************************************)
(

	eCycleDiagObj_Init						:= 0,
	eCycleDiagObj_ReadTemperature			,
	eCycleDiagObj_ReadErrorIndices			,	
	eCycleDiagObj_ReadDiag					,	
	eCycleDiagObj_ReadDelay					,	
	eCycleDiagObj_Done						,
	eCycleDiagObj_Error						:=999,
	eCycleDiagObj_NoError					
	
);
END_TYPE
(* End *)

// ---- DUTs/40_TwinSAFE/TwinSAFE_Connection/ST_TsConnectionInfo1Byte.TcDUT
TYPE ST_TsConnectionInfo1Byte :
(*******************************************************************************************************
Description			:	Connection information data of EtherCAT Slaves with 1 byte safe data 
Supported terminals : 	EL1904, EL2904...
Date 				:	04.04.2016
********************************************************************************************************)
STRUCT

	nState 	 								:USINT;
	nDiag 		 							:USINT;
	nInOutSafeDataByte1						:BYTE;
	
END_STRUCT
END_TYPE
(* End *)

// ---- DUTs/40_TwinSAFE/TwinSAFE_Connection/ST_TsConnectionInfo2Byte.TcDUT
TYPE ST_TsConnectionInfo2Byte :
(*******************************************************************************************************
Description			:	Connection information data of EtherCAT Slaves with 2 byte safe data 
Supported terminals : 	EK1914...
Date 				:	04.04.2016
********************************************************************************************************)
STRUCT

	nState 	 								:USINT;
	nDiag 		 							:USINT;
	nInOutSafeDataByte1						:BYTE;
	nInOutSafeDataByte2						:BYTE;
	
END_STRUCT
END_TYPE
(* End *)

// ---- DUTs/40_TwinSAFE/TwinSAFE_Connection/ST_TsConnectionInfo8Byte.TcDUT
TYPE ST_TsConnectionInfo8Byte :
(*******************************************************************************************************
Description			:	Connection information data of EtherCAT Slaves with 4 byte input and 4 byte output safe data  
Supported terminals : 	AX5805(2 Axis)
Date 				:	04.04.2016
********************************************************************************************************)
STRUCT

	nState  								:USINT;
	nDiag 	 								:USINT;
	nInSafeDataByte1						:BYTE;
	nInSafeDataByte2						:BYTE;
	nInSafeDataByte3						:BYTE;
	nInSafeDataByte4						:BYTE;
	nOutSafeDataByte1 						:BYTE;
	nOutSafeDataByte2 						:BYTE;
	nOutSafeDataByte3 						:BYTE;
	nOutSafeDataByte4 						:BYTE;

END_STRUCT
END_TYPE
(* End *)

// ---- DUTs/40_TwinSAFE/TwinSAFE_Connection/ST_TsConnectionInfoEL3214.TcDUT
TYPE ST_TsConnectionInfoEL3214 :
(*******************************************************************************************************
Description			:	Connection information data of EtherCAT Slave EL3214-0090 with 4 analog inputs  
Supported terminals : 	EL3214-0090
Date 				:	01.12.2016
********************************************************************************************************)
STRUCT

	nState  								:USINT;
	nDiag 	 								:USINT;
	nInSafeDataValue1						:INT;
	nInSafeDataValue2						:INT;
	nInSafeDataValue3						:INT;
	nInSafeDataValue4						:INT;

END_STRUCT
END_TYPE
(* End *)

// ---- DUTs/40_TwinSAFE/TwinSAFE_Connection/ST_TsConnectionInfoEL5021.TcDUT
TYPE ST_TsConnectionInfoEL5021 :
(*******************************************************************************************************
Description			:	Connection information data of EtherCAT Slave EL5021-0090 with 1 counter (1 Vss) input 
Supported terminals : 	EL5021-0090
Date 				:	01.12.2016
********************************************************************************************************)
STRUCT

	nState  								:USINT;
	nDiag 	 								:USINT;
	nInSafeDataCounterValue					:UDINT;
	nInSafeDataFrequencyValue				:DINT;
	nInSafeDataFrequencyValue16Bit			:INT;

END_STRUCT
END_TYPE
(* End *)

// ---- DUTs/40_TwinSAFE/TwinSAFE_Connection/ST_TsSlave2Temp.TcDUT
TYPE ST_TsSlave2Temp :
(*******************************************************************************************************
Description			:	EtherCAT Slaves with 2 internal temperatures
Supported terminals : 	EL1904, AX5805, AX5806
Date 				:	04.04.2016
********************************************************************************************************)
STRUCT

	nInternalTemperature1				:INT;	(* Temperature 1 [°C] *)
	nInternalTemperature2				:INT;	(* Temperature 2 [°C] *)
	
END_STRUCT
END_TYPE
(* End *)

// ---- DUTs/40_TwinSAFE/TwinSAFE_Connection/ST_TsSlave3Temp.TcDUT
TYPE ST_TsSlave3Temp :
(*******************************************************************************************************
Description			:	EtherCAT Slaves with 3 internal temperatures
Supported terminals : 	EL2904
Date 				:	04.04.2016
********************************************************************************************************)
STRUCT
	
	nInternalTemperature1					:INT;	(* Temperature 1 [°C] *)
	nInternalTemperature2					:INT;	(* Temperature 2 [°C] *)
	nInternalTemperatureOutputs				:INT;	(* Temperature 2 [°C] *)
	
END_STRUCT
END_TYPE
(* End *)

// ---- DUTs/40_TwinSAFE/TwinSAFE_Functionblocks/E_TsFbType.TcDUT
TYPE E_TsFbType :
(*******************************************************************************************************
Description			:	Enumeration TwinSAFE function block list
Documentation 		:	TwinSAFE-Logik-FB TwinCAT function blocks for TwinSAFE logic terminals
Supported hardware	: 	KL6904 / EL6900 / EL6910 / EJ6910 / EK1960
Version/Date 		:	V3.1.0/26.10.2016
********************************************************************************************************)
(
	
(* KL6904 / EL6900 / EL6910 / EJ6910 / EK1960 *)
	FB_TYPE_AND								:=0,
	FB_TYPE_OR								,
	FB_TYPE_OPMODE							,
	FB_TYPE_ESTOP							,
	FB_TYPE_MON								,
	FB_TYPE_DECOUPLER						,
	FB_TYPE_TWOHAND							,
	FB_TYPE_MUTING							,
	FB_TYPE_EDM								,
	FB_TYPE_RS								,
	FB_TYPE_SR								,
	FB_TYPE_TON								,
	FB_TYPE_TOF								,
	FB_TYPE_CONSHUT							,

(* only EL6910 / EJ6910 / EK1960 *)
	FB_TYPE_ADD								,
	FB_TYPE_SUB								,
	FB_TYPE_MUL								,
	FB_TYPE_DIV								,
	FB_TYPE_COMPARE							,
	FB_TYPE_LIMIT							,
	FB_TYPE_COUNTER							,
	FB_TYPE_SCALE							,
	FB_TYPE_SPEED							,
	FB_TYPE_LOADSENSING						,
	FB_TYPE_CAMMONITOR						,
	FB_TYPE_SLI								,
	FB_TYPE_ENVELOPE						,
	FB_TYPE_VIOLATIONCOUNTER				

);
END_TYPE
(* End *)

// ---- DUTs/40_TwinSAFE/TwinSAFE_Functionblocks/ST_TsFbInfo.TcDUT
TYPE ST_TsFbInfo :
STRUCT
	
	nState  								:USINT;
	nDiag  									:UINT;

END_STRUCT
END_TYPE
(* End *)

// ---- DUTs/40_TwinSAFE/TwinSAFE_Group/ST_TsGroupInfo.TcDUT
TYPE ST_TsGroupInfo :
STRUCT

	nState	 	 							:USINT;
	nDiag 	 								:USINT;

END_STRUCT
END_TYPE
(* End *)

// ---- DUTs/E_SampleMode.TcDUT
TYPE E_SampleMode :
(
	eSMode_Idle,
	eSMode_MC2_Req,
	eSMode_MC2_Act,
	eSMode_NCI_Req,
	eSMode_NCI_Act,
	eSMode_OOP_Req,
	eSMode_OOP_Act,
	eSMode_OOPConv_Req,
	eSMode_OOPConv_Act,
	eSMode_Last
);
END_TYPE

// ---- POUs/Database Server/E_WriteMode.TcDUT
{attribute 'qualified_only'}
{attribute 'strict'}
TYPE E_WriteMode :
(
	ePLCDBCmd   := 0,
	ePLCDBWriteStruct	:= 1,
	ePLCDBReadStruct 	:= 2
	
);
END_TYPE

// ---- POUs/Database Server/ST_CSVDataStruct.TcDUT
TYPE ST_CSVDataStruct :
STRUCT
	ID: LINT;
	Timestamp: DT;
	Name: STRING(80);
	Velocity: LREAL;
	Temperature: LREAL;
END_STRUCT
END_TYPE

// ---- POUs/IoT and JsonXml/IoTDataStruct.TcDUT
TYPE IoTDataStruct :
STRUCT
	{attribute 'iot.DisplayName' := 'Pulse 1'}
	{attribute 'iot.ReadOnly' := 'TRUE'}
	Puls1		:REAL;
	
	{attribute 'iot.DisplayName' := 'Pulse 2'}
	{attribute 'iot.ReadOnly' := 'TRUE'}
	Puls2	 	: REAL;
	
	{attribute 'iot.DisplayName' := 'Sinus Slow'}
	{attribute 'iot.ReadOnly' := 'TRUE'}
	Sinus_Slow 	: REAL;
	
	{attribute 'iot.DisplayName' := 'Generate Data'}
	bGenerateData : BOOL := TRUE;
	
	{attribute 'iot.DisplayName' := 'Reset Data'}
	bClearValues 	: BOOL;
END_STRUCT
END_TYPE

// ---- POUs/Sample OOP/Regulator/ST_RegParams.TcDUT
TYPE ST_RegParams : 
STRUCT
	fCtrlCycleTime	 : LREAL;
	fKp		 : LREAL;
	fTn		 : LREAL;
	fTv		 : LREAL;
	fTd		 : LREAL;
END_STRUCT
END_TYPE

// ---- POUs/Sample OOP/Table/E_AxisState.TcDUT
TYPE E_AxisState :
(
	eAxisState_Idle,
	eAxisState_Diag,
	eAxisState_Move,
	eAxisState_Reset
);
END_TYPE

// ---- POUs/Sample OOP/Table/E_MoveCmd.TcDUT
TYPE E_MoveCmd :
(
	eCmd_Idle,
	eCmd_MoveAbsolute,
	eCmd_MoveModulo,
	eCmd_MoveRelative,
	eCmd_MoveVelocity
);
END_TYPE

// ---- POUs/Sample OOP Conveyor/Device And Station Blocks/Internal/E_Modes.TcDUT
TYPE E_Modes :
(
	E_Disabled 			:= 0,
	E_Error 			:= 1,
	E_Manual 			:= 2,
	E_Auto 				:= 3,
	E_Reset 			:= 4,
	E_Resetting 		:= 5,
	E_SwitchingToAuto 	:= 6,
	E_SwitchingToManual := 7
);
END_TYPE

// ---- POUs/Sample OOP Conveyor/Device And Station Blocks/Internal/E_PartQuality.TcDUT
TYPE E_PartQuality :
(
	eRejected 	:= 0,
	eLow 		:= 1,
	eMid 		:= 2, 
	eHigh 		:= 3
);
END_TYPE

// ---- POUs/Sample OOP Conveyor/Device And Station Blocks/Internal/ST_PartData.TcDUT
TYPE ST_PartData :
STRUCT
	iIDNumber 					: UDINT; // ID Number of the part 
	iCurrentDeviceID 			: UDINT; // ID of the current device that contains the part eg station1
	iSubDeviceLocation 			: UDINT; // Sublocation if available eg bin number within a station
	fPosition 					: LREAL; // Current position within a device eg conveyor location  
	fLength 					: LREAL; // length of part
	fStartingConveyorPosition	: LREAL; // conveyor position when product was placed
END_STRUCT
END_TYPE

// ---- POUs/SampleIEC Languages/Datatypes/E_Commands.TcDUT
TYPE E_Commands :
(
		eCommandIdle := 0,
		eCommandRun,
		eCommandStop
);
END_TYPE

// ---- POUs/SampleIEC Languages/Datatypes/E_Operation.TcDUT
TYPE E_Operation :
(
	eOp_Add := 0,
	eOp_Sub,
	eOp_Mul
);
END_TYPE

// ---- GVLs/GVL.TcGVL
VAR_GLOBAL CONSTANT
	iMAX_AXES_REF : INT := 5;
END_VAR
VAR_GLOBAL
	iGlobalCounter : UINT;
	fbCrititcalSection : FB_IecCriticalSection;
END_VAR

// ---- GVLs/GVL00_IO_CX.TcGVL
(* GVL00_IO_CX *)
{attribute 'TcContextName' := 'PlcTask'}
VAR_GLOBAL

	(* EL1008 digital inputs *)
	bSwitchS10						AT%I*	:BOOL;	(* blinker 1 on/off *)
	bSwitchS11						AT%I*	:BOOL;	(* blinker 2 on/off *)
	bSwitchS12						AT%I*	:BOOL;	(* controller enable axis 1 *)
	bSwitchS13						AT%I*	:BOOL;	(* controller enable axis 2 *)
	bSwitchS14						AT%I*	:BOOL;	(* controller enable axis 3 *)
	bSwitchS15						AT%I*	:BOOL;	(* controller enable Axis 4 *)
	bSwitchS16						AT%I*	:BOOL;	(* start axis 1 - 4 absolute *)
	bSwitchS17						AT%I*	:BOOL;	(* Uncouple Axis 1 - 4 / set target position to zero *)
	
	(* EL2008 digital outputs *)
	bLedH10							AT%Q*	:BOOL;	(* blinker 1 *)
	bLedH11							AT%Q*	:BOOL;	(* blinker 2 *)
	bLedH12							AT%Q*	:BOOL;	(* axis 1 operational *)
	bLedH13							AT%Q*	:BOOL;	(* axis 2 operational *)
	bLedH14							AT%Q*	:BOOL;	(* axis 3 operational *)
	bLedH15							AT%Q*	:BOOL;	(* axis 4 operational *)
	bLedH16							AT%Q*	:BOOL;	(* bSwitchS16 aktiv *)
	bLedH17							AT%Q*	:BOOL;	(* bSwitchS17 aktiv *)

	(* EL5151 incremental encoder 24 increments/rotation * 4-fold evaluation -> 96  increments/rotation*)
	nHandwheelCounter				AT%I*	:UINT;	(* handwheel counter (Axis_5_Encoder) *)
	bHandwheelSwitchS28				AT%I*	:BOOL;	(* axis 1 - 4 couple to the handwheel *)	

	(* EL9110 potential supply diagnosis *)
	bPotentialStepper24VOk			AT%I*	:BOOL;	(* Power stepper ok *)

	(* EL9576 brake chopper terminal *)
	
	(* EL7037 (Axis 1 Stepper) stepper motor terminal inputs *)
	bStepperReferenceCam 			AT%I*	:BOOL;	(* stepper reference cam (Axis 1 Stepper) *)
	bSwitchS23						AT%I*	:BOOL;	(* start stepper homing *)
	bSwitchS24						AT%I*	:BOOL;	(*  *)	

	(* EL9512 power supply diagnosis *)
	bPotentialAnalog12VOk			AT%I*	:BOOL;	(* 12V voltage ok *)
	
	(* EL3162 0..10V analog inputs *)
	nAnalogInR10					AT%I*	:INT;	(* override axis 1 - 2, blinker 1 *)
	nAnalogInFromEL4102Out1			AT%I*	:INT;	(* *)

	(* EL4102 0..10V analog outputs *)
	nAnalogOutP10					AT%Q*	:INT;	(* Override axis 1 - 2 / 10.0V = 100% *)
{attribute 'TcContextName' := 'PlcTaskFast'}
	nAnalogOutP11					AT%Q*	:INT;	(* Override axis 3 - 4 / 10.0V = 100% *)

	(* EL6900 TwinSAFE Logic *)

END_VAR
(* End *)

// ---- GVLs/GVL01_IO_EK1100.TcGVL
(* GVL01_IO_EK1100 *)
{attribute 'TcContextName' := 'PlcTask'}
VAR_GLOBAL

	(* EL1859 digital inputs/outputs *)
	bSwitchS20						AT%I*	:BOOL;	(* Start sequence axis 1-4 *)
	bSwitchS21						AT%I*	:BOOL;	(* Reset axis 1-4 *)
	bSwitchS22						AT%I*	:BOOL;	(* not in use *)
	bSwitchS31						AT%I*	:BOOL;	(* Error acknowledge / reset Axis 1 - 4 *)
	bAxis2ReferenceCamEL1			AT%I*	:BOOL;	(* servo reference cam on a standard input (Axis 2 Servo EL) *)

	bLedH31							AT%Q*	:BOOL;	(* Led reset button *)
	bLedH32							AT%Q*	:BOOL;	(* S32 aktiv *)
	bLedH33							AT%Q*	:BOOL;	(* S33 aktiv *)

	bLedH23							AT%Q*	:BOOL;	(* stepper homing done *)
	bLedH24							AT%Q*	:BOOL;	(* not in use *)
	bLedH25							AT%Q*	:BOOL;	(* Modulo touch probe aktiv *)
	bLedH26							AT%Q*	:BOOL;	(* Reference cam axis 3 *)

	(* EL1904 digital inputs TwinSAFE *)
	
	(* EL2904 digital outputs TwinSAFE *)	
	
	(* EL9110 potential supply diagnosis switched from the contactor -K1 (TwinSAFE) *)
	bPotentialConduktorK124VOk		AT%I*	:BOOL;	(* Power on *)
	
	(* EL2004 digital outputs *)
	bLedH20							AT%Q*	:BOOL;	(* Sequence axis 1-4 busy (flashes) *)
	bLedH21							AT%Q*	:BOOL;	(* Error axis 1-4 (flashes) *)
	bLedH22							AT%Q*	:BOOL;	(* not in use *)

	(* EL9410 potential supply diagnosis *)
	bPotentialEBusUs24VNotOk		AT%I*	:BOOL;	(* E-BUS power not ok *)
	bPotentialServoUp24VNotOk		AT%I*	:BOOL;	(* Power servo (EL7201) not ok *)

	(* EL7201 (Axis 2 Servo EL) servomotor terminal inputs *)
	bAxis2ReferenceCamEL7 			AT%I*	:BOOL;	(* servo reference cam on the EL7201 input (Axis 2 Servo EL) *)
	bSwitchS25						AT%I*	:BOOL;	(* Modulo touch probe on *)
	nAxis2ActTorque					AT%I*	:INT;	(* axis 2 current +/- 1000 *)

END_VAR
(* End *)

// ---- GVLs/GVL02_IO_EK1101.TcGVL
(* GVL02_IO_EK1101 *)
{attribute 'TcContextName' := 'PlcTask'}
VAR_GLOBAL
	
	(* EL1904 digital inputs TwinSAFE *)

	(* EL1252 digital inputs time stamp *)
	stEL1252Ch1								:EL1252_IoInterface;	(* servo reference cam on a time stamp input (axis 2 servo EL) *)
	stEL1252Ch2								:EL1252_IoInterface;	(* Signal form EL2252 output 1 *)

	(* EL1262 digital inputs oversampling *)
	nEL1262Ch1CycleCount			AT%I*	:UINT;					(* EtherCAT cycle count, increments each EtherCAT cycle *)
	aAxis2RefCamOs		 			AT%I*	:ARRAY[0..9] OF BOOL;	(* servo reference cam on a oversampling input (Axis 2 Servo EL) - Oversampling of 10 samples per EtherCAT cylce (based on task cylce time) *)
	nEL1262Ch2CycleCount			AT%I*	:UINT;					(* EtherCAT cycle count, increments each EtherCAT cycle *)
	aOsInputFromEL2252Out2			AT%I*	:ARRAY[0..9] OF BOOL;	(* Signal form EL2252 output 2 - Oversampling of 10 samples per EtherCAT cylce (based on task cylce time) *)

	(* EL2252 digital outputs time stamp *)
	stEL2252								:EL2252_IoInterface;	(* Ch1 - position cam axis 2  90 - 180 Degree
																   	   Ch2 - position cam axis 2  30 - 90  Degree *)
	
	(* EL3702 analog inputs oversampling *)
	nEL3702Ch1CycleCount			AT%I*	:UINT;					(* EtherCAT cycle count, increments each EtherCAT cycle *)
{attribute 'TcContextName' := 'PlcTaskFast'}
	aOsAnalogInR11		 			AT%I*	:ARRAY[0..9] OF INT;	(* override axis 3 - 4 - Oversampling of 10 samples per EtherCAT cylce (based on task cylce time) *)
	nEL3702Ch2CycleCount			AT%I*	:UINT;					(* EtherCAT cycle count, increments each EtherCAT cycle *)
{attribute 'TcContextName' := 'PlcTaskFast'}
	aOsInputFromEL4732Out1 			AT%I*	:ARRAY[0..9] OF INT;	(* Signal form EL4732 output 1 - Oversampling of 10 samples per EtherCAT cylce (based on task cylce time) *)
	
	(* EL4732 analog outputs oversampling *)
	nEL4732Ch1CycleCount			AT%Q*	:UINT;					(* EtherCAT cycle count, increments each EtherCAT cycle *)
	aOsOutputToEL3702In2 			AT%Q*	:ARRAY[0..99] OF INT;	(* Signal to EL3702 input 2 - Oversampling of 100 samples per EtherCAT cylce (based on task cylce time) *)
	
	(* EL2004 digital outputs *)
	
END_VAR
(* End *)

